KUKA KRL program: filwin69start.src

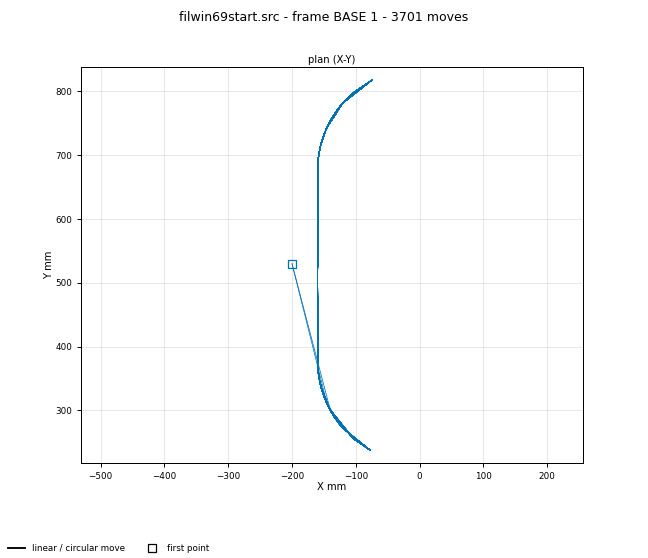
[picture p0: tool path of filwin69start.src in frame BASE 1, 3701 of 3702 moves have a stored position in this frame; points joined in program order, loops and branches not executed]
&ACCESS RVEO
&REL 11
&PARAM TEMPLATE = C:\KRC\Roboter\Template\vorgabe
&PARAM EDITMASK = *
DEF variable_helical2( )
;FOLD INI
  ;FOLD BASISTECH INI
    GLOBAL INTERRUPT DECL 3 WHEN $STOPMESS==TRUE DO IR_STOPM ( )
    INTERRUPT ON 3
    BAS (#INITMOV,0 )
  ;ENDFOLD (BASISTECH INI)
 ;FOLD USER INI


    ;Make your modifications here
  ;ENDFOLD (USER INI)
;ENDFOLD (INI)
ACTION(#AXIS_RESET,34,1000,#NOERROR,ERROR_CODE)
;FOLD PTP HOME  Vel= 100 % DEFAULT;%{PE}%MKUKATPBASIS,%CMOVE,%VPTP,%P 1:PTP, 2:HOME, 3:, 5:100, 7:DEFAULT
$BWDSTART = FALSE
PDAT_ACT=PDEFAULT
FDAT_ACT=FHOME
BAS (#PTP_PARAMS,100 )
$H_POS=XHOME
PTP  XHOME
;ENDFOLD
BAS(#TOOL,1)
BAS(#BASE,1)
$VEL_AXIS[1]=100
$VEL_AXIS[2]=100
$VEL_AXIS[3]=100
$VEL_AXIS[4]=100
$VEL_AXIS[5]=100
$VEL_AXIS[6]=100
$VEL_EXTAX[1]=100
$VEL_EXTAX[2]=100

$ACC_AXIS[1]=100
$ACC_AXIS[2]=100
$ACC_AXIS[3]=100
$ACC_AXIS[4]=100
$ACC_AXIS[5]=100
$ACC_AXIS[6]=100
$ACC_EXTAX[1]=100
$ACC_EXTAX[2]=100

;;;;;;;;; postprocessing parameters (date 2024-01-29T17:39:48.607859)
; qxconst: -159.99
; qxconstarcys: -152.5,146.5
; qE3offset: 0.00
; qyoffset: 530.00
; qswitchsplit: 3
; qthinningtol: 0.2010
;;;;;;;;;

SLIN {X  -200.000, Y  +530.000, Z    +0.000, A    +0.000, E1    +0.000, E3    +0.000, E4    +0.000}

SLIN {X  -139.652, Y  +299.435, Z    +0.000, E1   +73.041, E3  -288.222}
HALT
SPLINE
SPL {X  -136.475, Y  +294.006, Z    +0.000, E1   +72.670, E3  -282.347}
SPL {X  -133.214, Y  +288.895, Z    +0.000, E1   +72.272, E3  -276.699}
SPL {X  -129.829, Y  +284.006, Z    +0.000, E1   +71.844, E3  -271.224}
SPL {X  -126.314, Y  +279.309, Z    +0.000, E1   +71.374, E3  -265.932}
SPL {X  -122.705, Y  +274.834, Z    +0.000, E1   +70.869, E3  -260.920}
SPL {X  -119.804, Y  +271.463, Z    +0.000, E1   +70.429, E3  -257.202}
SPL {X   -77.409, Y  +237.483, Z    +0.000, E1   +59.013, E3  -163.526}
ENDSPLINE

SPLINE
SPL {X  -103.775, Y  +255.731, Z    +0.000, E1   +56.205, E3   +33.187}
SPL {X  -133.021, Y  +288.605, Z    +0.000, E1   +53.007, E3   +64.644}
SPL {X  -149.384, Y  +320.219, Z    +0.000, E1   +43.953, E3   +76.367}
SPL {X  -157.534, Y  +349.577, Z    +0.000, E1   +27.748, E3   +81.719}
SPL {X  -159.460, Y  +364.489, Z    +0.000, E1   +15.407, E3   +83.014}
SPL {X  -159.962, Y  +374.520, Z    +0.000, E1    +5.534, E3   +83.410}
SPL {X  -159.990, Y  +379.490, Z    +0.000, E1    +0.023, E3   +83.468}
SPL {X  -159.990, Y  +381.667, Z    +0.000, E1    -4.707, E3   +83.490}
SPL {X  -159.990, Y  +387.434, Z    +0.000, E1   -19.600, E3   +83.672}
SPL {X  -159.990, Y  +392.971, Z    +0.000, E1   -33.903, E3   +84.005}
SPL {X  -159.990, Y  +399.006, Z    +0.000, E1   -45.565, E3   +84.581}
SPL {X  -159.990, Y  +410.008, Z    +0.000, E1   -58.546, E3   +86.192}
SPL {X  -159.990, Y  +426.664, Z    +0.000, E1   -66.963, E3   +89.813}
SPL {X  -159.990, Y  +494.829, Z    +0.000, E1   -73.764, E3  +111.577}
SPL {X  -158.798, Y  +695.991, Z    +0.000, E1   -74.986, E3  +201.510}
SPL {X  -156.512, Y  +709.677, Z    +0.000, E1   -74.772, E3  +211.653}
SPL {X  -153.684, Y  +720.975, Z    +0.000, E1   -74.508, E3  +220.940}
SPL {X  -149.353, Y  +733.863, Z    +0.000, E1   -74.100, E3  +232.528}
SPL {X  -145.190, Y  +743.705, Z    +0.000, E1   -73.640, E3  +242.209}
SPL {X  -141.940, Y  +750.322, Z    +0.000, E1   -73.290, E3  +248.976}
SPL {X  -138.555, Y  +756.496, Z    +0.000, E1   -72.905, E3  +255.541}
SPL {X  -135.025, Y  +762.319, Z    +0.000, E1   -72.483, E3  +261.921}
SPL {X  -131.747, Y  +767.272, Z    +0.000, E1   -72.071, E3  +267.446}
SPL {X  -128.648, Y  +771.613, Z    +0.000, E1   -71.666, E3  +272.338}
SPL {X  -125.012, Y  +776.344, Z    +0.000, E1   -71.184, E3  +277.650}
SPL {X  -121.578, Y  +780.498, Z    +0.000, E1   -70.681, E3  +282.293}
SPL {X  -119.460, Y  +782.925, Z    +0.000, E1   -70.353, E3  +284.957}
SPL {X   -74.295, Y  +818.193, Z    +0.000, E1   -57.793, E3  +393.618}
ENDSPLINE

SPLINE
SPL {X  -120.240, Y  +782.043, Z    +0.000, E1   -55.019, E3  +592.114}
SPL {X  -145.777, Y  +742.423, Z    +0.000, E1   -46.722, E3  +613.993}
SPL {X  -154.920, Y  +716.458, Z    +0.000, E1   -35.175, E3  +620.048}
SPL {X  -159.063, Y  +693.702, Z    +0.000, E1   -19.028, E3  +622.830}
SPL {X  -159.958, Y  +679.684, Z    +0.000, E1    -5.688, E3  +623.541}
SPL {X  -159.990, Y  +674.512, Z    +0.000, E1    -0.026, E3  +623.606}
SPL {X  -159.990, Y  +672.767, Z    +0.000, E1    +3.705, E3  +623.619}
SPL {X  -159.990, Y  +669.310, Z    +0.000, E1   +12.444, E3  +623.693}
SPL {X  -159.990, Y  +665.511, Z    +0.000, E1   +22.359, E3  +623.852}
SPL {X  -159.990, Y  +658.432, Z    +0.000, E1   +38.720, E3  +624.377}
SPL {X  -159.990, Y  +646.280, Z    +0.000, E1   +56.156, E3  +625.906}
SPL {X  -159.990, Y  +625.549, Z    +0.000, E1   +67.208, E3  +630.427}
SPL {X  -159.990, Y  +550.186, Z    +0.000, E1   +73.637, E3  +655.833}
SPL {X  -159.493, Y  +364.902, Z    +0.000, E1   +74.541, E3  +742.826}
SPL {X  -156.915, Y  +346.281, Z    +0.000, E1   +74.304, E3  +756.422}
ENDSPLINE

SPLINE
SPL {X  -159.697, Y  +367.814, Z    +0.000, E1   +71.217, E3  +773.741}
ENDSPLINE

SPLINE
SPL {X  -157.536, Y  +349.586, Z    +0.000, E1   +71.787, E3  +781.039}
SPL {X  -154.855, Y  +337.291, Z    +0.000, E1   +72.155, E3  +785.793}
SPL {X  -150.925, Y  +324.412, Z    +0.000, E1   +72.419, E3  +791.687}
SPL {X  -146.819, Y  +313.931, Z    +0.000, E1   +72.621, E3  +796.380}
SPL {X  -140.820, Y  +301.561, Z    +0.000, E1   +73.023, E3  +800.297}
SPL {X  -136.475, Y  +294.006, Z    +0.000, E1   +72.670, E3  +807.206}
SPL {X  -133.214, Y  +288.895, Z    +0.000, E1   +72.272, E3  +812.853}
SPL {X  -129.829, Y  +284.006, Z    +0.000, E1   +71.844, E3  +818.328}
SPL {X  -126.314, Y  +279.309, Z    +0.000, E1   +71.374, E3  +823.621}
SPL {X  -122.705, Y  +274.834, Z    +0.000, E1   +70.869, E3  +828.632}
SPL {X  -119.804, Y  +271.463, Z    +0.000, E1   +70.429, E3  +832.351}
SPL {X   -77.409, Y  +237.483, Z    +0.000, E1   +59.013, E3  +926.026}
ENDSPLINE

SPLINE
SPL {X  -103.775, Y  +255.731, Z    +0.000, E1   +56.205, E3 +1122.739}
SPL {X  -141.196, Y  +302.265, Z    +0.000, E1   +49.914, E3 +1160.224}
SPL {X  -155.405, Y  +339.473, Z    +0.000, E1   +34.418, E3 +1169.925}
SPL {X  -159.172, Y  +361.346, Z    +0.000, E1   +18.323, E3 +1172.349}
SPL {X  -159.962, Y  +374.520, Z    +0.000, E1    +5.534, E3 +1172.962}
SPL {X  -159.990, Y  +379.490, Z    +0.000, E1    +0.023, E3 +1173.020}
SPL {X  -159.990, Y  +381.667, Z    +0.000, E1    -4.707, E3 +1173.042}
SPL {X  -159.990, Y  +385.814, Z    +0.000, E1   -15.621, E3 +1173.146}
SPL {X  -159.990, Y  +390.948, Z    +0.000, E1   -28.850, E3 +1173.422}
SPL {X  -159.990, Y  +399.006, Z    +0.000, E1   -45.565, E3 +1174.134}
SPL {X  -159.990, Y  +410.008, Z    +0.000, E1   -58.546, E3 +1175.744}
SPL {X  -159.990, Y  +426.664, Z    +0.000, E1   -66.963, E3 +1179.365}
SPL {X  -159.990, Y  +494.829, Z    +0.000, E1   -73.764, E3 +1201.129}
SPL {X  -158.798, Y  +695.991, Z    +0.000, E1   -74.986, E3 +1291.062}
SPL {X  -156.512, Y  +709.677, Z    +0.000, E1   -74.772, E3 +1301.205}
SPL {X  -153.684, Y  +720.975, Z    +0.000, E1   -74.508, E3 +1310.493}
SPL {X  -149.353, Y  +733.863, Z    +0.000, E1   -74.100, E3 +1322.080}
SPL {X  -145.190, Y  +743.705, Z    +0.000, E1   -73.640, E3 +1331.761}
SPL {X  -141.940, Y  +750.322, Z    +0.000, E1   -73.290, E3 +1338.528}
SPL {X  -138.555, Y  +756.496, Z    +0.000, E1   -72.905, E3 +1345.093}
SPL {X  -135.025, Y  +762.319, Z    +0.000, E1   -72.483, E3 +1351.473}
SPL {X  -131.747, Y  +767.272, Z    +0.000, E1   -72.071, E3 +1356.998}
SPL {X  -128.648, Y  +771.613, Z    +0.000, E1   -71.666, E3 +1361.890}
SPL {X  -125.012, Y  +776.344, Z    +0.000, E1   -71.184, E3 +1367.202}
SPL {X  -121.578, Y  +780.498, Z    +0.000, E1   -70.681, E3 +1371.845}
SPL {X  -119.460, Y  +782.925, Z    +0.000, E1   -70.353, E3 +1374.509}
SPL {X   -74.295, Y  +818.193, Z    +0.000, E1   -57.793, E3 +1483.170}
ENDSPLINE

SPLINE
SPL {X  -120.240, Y  +782.043, Z    +0.000, E1   -55.019, E3 +1681.666}
SPL {X  -145.777, Y  +742.423, Z    +0.000, E1   -46.722, E3 +1703.545}
SPL {X  -154.920, Y  +716.458, Z    +0.000, E1   -35.175, E3 +1709.600}
SPL {X  -159.063, Y  +693.702, Z    +0.000, E1   -19.028, E3 +1712.382}
SPL {X  -159.958, Y  +679.684, Z    +0.000, E1    -5.688, E3 +1713.094}
SPL {X  -159.990, Y  +674.512, Z    +0.000, E1    -0.026, E3 +1713.158}
SPL {X  -159.990, Y  +672.767, Z    +0.000, E1    +3.705, E3 +1713.172}
SPL {X  -159.990, Y  +669.310, Z    +0.000, E1   +12.444, E3 +1713.246}
SPL {X  -159.990, Y  +665.511, Z    +0.000, E1   +22.359, E3 +1713.404}
SPL {X  -159.990, Y  +658.432, Z    +0.000, E1   +38.720, E3 +1713.929}
SPL {X  -159.990, Y  +646.280, Z    +0.000, E1   +56.156, E3 +1715.458}
SPL {X  -159.990, Y  +625.549, Z    +0.000, E1   +67.208, E3 +1719.979}
SPL {X  -159.990, Y  +550.186, Z    +0.000, E1   +73.637, E3 +1745.385}
SPL {X  -159.493, Y  +364.902, Z    +0.000, E1   +74.541, E3 +1832.378}
SPL {X  -156.915, Y  +346.281, Z    +0.000, E1   +74.304, E3 +1845.974}
ENDSPLINE

SPLINE
SPL {X  -159.697, Y  +367.814, Z    +0.000, E1   +71.217, E3 +1863.293}
ENDSPLINE

SPLINE
SPL {X  -157.536, Y  +349.586, Z    +0.000, E1   +71.787, E3 +1870.591}
SPL {X  -154.855, Y  +337.291, Z    +0.000, E1   +72.155, E3 +1875.345}
SPL {X  -150.925, Y  +324.412, Z    +0.000, E1   +72.419, E3 +1881.239}
SPL {X  -146.819, Y  +313.931, Z    +0.000, E1   +72.621, E3 +1885.933}
SPL {X  -140.820, Y  +301.561, Z    +0.000, E1   +73.023, E3 +1889.849}
SPL {X  -136.475, Y  +294.006, Z    +0.000, E1   +72.670, E3 +1896.758}
SPL {X  -133.214, Y  +288.895, Z    +0.000, E1   +72.272, E3 +1902.406}
SPL {X  -129.829, Y  +284.006, Z    +0.000, E1   +71.844, E3 +1907.881}
SPL {X  -126.314, Y  +279.309, Z    +0.000, E1   +71.374, E3 +1913.173}
SPL {X  -122.705, Y  +274.834, Z    +0.000, E1   +70.869, E3 +1918.184}
SPL {X  -119.804, Y  +271.463, Z    +0.000, E1   +70.429, E3 +1921.903}
SPL {X   -77.409, Y  +237.483, Z    +0.000, E1   +59.013, E3 +2015.578}
ENDSPLINE

SPLINE
SPL {X  -103.775, Y  +255.731, Z    +0.000, E1   +56.205, E3 +2212.292}
SPL {X  -141.196, Y  +302.265, Z    +0.000, E1   +49.914, E3 +2249.777}
SPL {X  -155.405, Y  +339.473, Z    +0.000, E1   +34.418, E3 +2259.477}
SPL {X  -159.172, Y  +361.346, Z    +0.000, E1   +18.323, E3 +2261.902}
SPL {X  -159.962, Y  +374.520, Z    +0.000, E1    +5.534, E3 +2262.515}
SPL {X  -159.990, Y  +379.490, Z    +0.000, E1    +0.023, E3 +2262.572}
SPL {X  -159.990, Y  +381.667, Z    +0.000, E1    -4.707, E3 +2262.594}
SPL {X  -159.990, Y  +385.814, Z    +0.000, E1   -15.621, E3 +2262.698}
SPL {X  -159.990, Y  +390.948, Z    +0.000, E1   -28.850, E3 +2262.974}
SPL {X  -159.990, Y  +399.006, Z    +0.000, E1   -45.565, E3 +2263.686}
SPL {X  -159.990, Y  +410.008, Z    +0.000, E1   -58.546, E3 +2265.296}
SPL {X  -159.990, Y  +426.664, Z    +0.000, E1   -66.963, E3 +2268.917}
SPL {X  -159.990, Y  +494.829, Z    +0.000, E1   -73.764, E3 +2290.681}
SPL {X  -158.798, Y  +695.991, Z    +0.000, E1   -74.986, E3 +2380.614}
SPL {X  -156.512, Y  +709.677, Z    +0.000, E1   -74.772, E3 +2390.758}
SPL {X  -153.684, Y  +720.975, Z    +0.000, E1   -74.508, E3 +2400.045}
SPL {X  -150.879, Y  +729.719, Z    +0.000, E1   -74.224, E3 +2407.839}
SPL {X  -148.237, Y  +736.689, Z    +0.000, E1   -73.960, E3 +2414.393}
SPL {X  -145.190, Y  +743.705, Z    +0.000, E1   -73.640, E3 +2421.314}
SPL {X  -141.940, Y  +750.322, Z    +0.000, E1   -73.290, E3 +2428.081}
SPL {X  -138.555, Y  +756.496, Z    +0.000, E1   -72.905, E3 +2434.646}
SPL {X  -135.025, Y  +762.319, Z    +0.000, E1   -72.483, E3 +2441.025}
SPL {X  -131.747, Y  +767.272, Z    +0.000, E1   -72.071, E3 +2446.550}
SPL {X  -127.432, Y  +773.236, Z    +0.000, E1   -71.530, E3 +2453.236}
SPL {X  -124.036, Y  +777.554, Z    +0.000, E1   -71.026, E3 +2458.134}
SPL {X  -120.782, Y  +781.422, Z    +0.000, E1   -70.584, E3 +2462.392}
SPL {X   -74.295, Y  +818.193, Z    +0.000, E1   -57.793, E3 +2572.722}
ENDSPLINE

SPLINE
SPL {X  -105.102, Y  +797.125, Z    +0.000, E1   -55.734, E3 +2752.089}
SPL {X  -126.361, Y  +774.631, Z    +0.000, E1   -54.192, E3 +2777.757}
SPL {X  -145.777, Y  +742.423, Z    +0.000, E1   -46.722, E3 +2793.098}
SPL {X  -154.920, Y  +716.458, Z    +0.000, E1   -35.175, E3 +2799.153}
SPL {X  -159.063, Y  +693.702, Z    +0.000, E1   -19.028, E3 +2801.934}
SPL {X  -159.958, Y  +679.684, Z    +0.000, E1    -5.688, E3 +2802.646}
SPL {X  -159.990, Y  +674.512, Z    +0.000, E1    -0.026, E3 +2802.711}
SPL {X  -159.990, Y  +672.767, Z    +0.000, E1    +3.705, E3 +2802.724}
SPL {X  -159.990, Y  +669.310, Z    +0.000, E1   +12.444, E3 +2802.798}
SPL {X  -159.990, Y  +665.511, Z    +0.000, E1   +22.359, E3 +2802.957}
SPL {X  -159.990, Y  +660.776, Z    +0.000, E1   +34.018, E3 +2803.263}
SPL {X  -159.990, Y  +655.863, Z    +0.000, E1   +43.768, E3 +2803.721}
SPL {X  -159.990, Y  +646.280, Z    +0.000, E1   +56.156, E3 +2805.010}
SPL {X  -159.990, Y  +625.549, Z    +0.000, E1   +67.208, E3 +2809.532}
SPL {X  -159.990, Y  +550.186, Z    +0.000, E1   +73.637, E3 +2834.937}
SPL {X  -159.493, Y  +364.902, Z    +0.000, E1   +74.541, E3 +2921.931}
SPL {X  -156.915, Y  +346.281, Z    +0.000, E1   +74.304, E3 +2935.527}
ENDSPLINE

SPLINE
SPL {X  -159.697, Y  +367.814, Z    +0.000, E1   +71.217, E3 +2952.845}
ENDSPLINE

SPLINE
SPL {X  -157.536, Y  +349.586, Z    +0.000, E1   +71.787, E3 +2960.143}
SPL {X  -154.855, Y  +337.291, Z    +0.000, E1   +72.155, E3 +2964.897}
SPL {X  -150.925, Y  +324.412, Z    +0.000, E1   +72.419, E3 +2970.792}
SPL {X  -146.819, Y  +313.931, Z    +0.000, E1   +72.621, E3 +2975.485}
SPL {X  -140.820, Y  +301.561, Z    +0.000, E1   +73.023, E3 +2979.401}
SPL {X  -136.475, Y  +294.006, Z    +0.000, E1   +72.670, E3 +2986.310}
SPL {X  -133.214, Y  +288.895, Z    +0.000, E1   +72.272, E3 +2991.958}
SPL {X  -129.829, Y  +284.006, Z    +0.000, E1   +71.844, E3 +2997.433}
SPL {X  -126.314, Y  +279.309, Z    +0.000, E1   +71.374, E3 +3002.725}
SPL {X  -122.705, Y  +274.834, Z    +0.000, E1   +70.869, E3 +3007.736}
SPL {X  -119.804, Y  +271.463, Z    +0.000, E1   +70.429, E3 +3011.455}
SPL {X   -77.409, Y  +237.483, Z    +0.000, E1   +59.013, E3 +3105.131}
ENDSPLINE

SPLINE
SPL {X  -103.775, Y  +255.731, Z    +0.000, E1   +56.205, E3 +3301.844}
SPL {X  -141.196, Y  +302.265, Z    +0.000, E1   +49.914, E3 +3339.329}
SPL {X  -155.405, Y  +339.473, Z    +0.000, E1   +34.418, E3 +3349.029}
SPL {X  -159.172, Y  +361.346, Z    +0.000, E1   +18.323, E3 +3351.454}
SPL {X  -159.962, Y  +374.520, Z    +0.000, E1    +5.534, E3 +3352.067}
SPL {X  -159.990, Y  +379.490, Z    +0.000, E1    +0.023, E3 +3352.124}
SPL {X  -159.990, Y  +381.667, Z    +0.000, E1    -4.707, E3 +3352.146}
SPL {X  -159.990, Y  +387.434, Z    +0.000, E1   -19.600, E3 +3352.329}
SPL {X  -159.990, Y  +395.000, Z    +0.000, E1   -38.121, E3 +3352.838}
SPL {X  -159.990, Y  +406.380, Z    +0.000, E1   -55.108, E3 +3354.279}
SPL {X  -159.990, Y  +426.664, Z    +0.000, E1   -66.963, E3 +3358.469}
SPL {X  -159.990, Y  +494.829, Z    +0.000, E1   -73.764, E3 +3380.234}
SPL {X  -158.798, Y  +695.991, Z    +0.000, E1   -74.986, E3 +3470.166}
SPL {X  -156.512, Y  +709.677, Z    +0.000, E1   -74.772, E3 +3480.310}
SPL {X  -153.684, Y  +720.975, Z    +0.000, E1   -74.508, E3 +3489.597}
SPL {X  -149.353, Y  +733.863, Z    +0.000, E1   -74.100, E3 +3501.185}
SPL {X  -145.190, Y  +743.705, Z    +0.000, E1   -73.640, E3 +3510.866}
SPL {X  -141.940, Y  +750.322, Z    +0.000, E1   -73.290, E3 +3517.633}
SPL {X  -138.555, Y  +756.496, Z    +0.000, E1   -72.905, E3 +3524.198}
SPL {X  -135.025, Y  +762.319, Z    +0.000, E1   -72.483, E3 +3530.577}
SPL {X  -131.747, Y  +767.272, Z    +0.000, E1   -72.071, E3 +3536.102}
SPL {X  -127.432, Y  +773.236, Z    +0.000, E1   -71.530, E3 +3542.788}
SPL {X  -124.036, Y  +777.554, Z    +0.000, E1   -71.026, E3 +3547.686}
SPL {X  -120.782, Y  +781.422, Z    +0.000, E1   -70.584, E3 +3551.944}
SPL {X   -74.295, Y  +818.193, Z    +0.000, E1   -57.793, E3 +3662.275}
ENDSPLINE

SPLINE
SPL {X  -105.102, Y  +797.125, Z    +0.000, E1   -55.734, E3 +3841.641}
SPL {X  -126.361, Y  +774.631, Z    +0.000, E1   -54.192, E3 +3867.309}
SPL {X  -145.777, Y  +742.423, Z    +0.000, E1   -46.722, E3 +3882.650}
SPL {X  -154.920, Y  +716.458, Z    +0.000, E1   -35.175, E3 +3888.705}
SPL {X  -159.063, Y  +693.702, Z    +0.000, E1   -19.028, E3 +3891.486}
SPL {X  -159.958, Y  +679.684, Z    +0.000, E1    -5.688, E3 +3892.198}
SPL {X  -159.990, Y  +674.512, Z    +0.000, E1    -0.026, E3 +3892.263}
SPL {X  -159.990, Y  +672.767, Z    +0.000, E1    +3.705, E3 +3892.276}
SPL {X  -159.990, Y  +669.310, Z    +0.000, E1   +12.444, E3 +3892.350}
SPL {X  -159.990, Y  +665.511, Z    +0.000, E1   +22.359, E3 +3892.509}
SPL {X  -159.990, Y  +660.776, Z    +0.000, E1   +34.018, E3 +3892.815}
SPL {X  -159.990, Y  +655.863, Z    +0.000, E1   +43.768, E3 +3893.273}
SPL {X  -159.990, Y  +646.280, Z    +0.000, E1   +56.156, E3 +3894.562}
SPL {X  -159.990, Y  +625.549, Z    +0.000, E1   +67.208, E3 +3899.084}
SPL {X  -159.990, Y  +550.186, Z    +0.000, E1   +73.637, E3 +3924.490}
SPL {X  -159.493, Y  +364.902, Z    +0.000, E1   +74.541, E3 +4011.483}
SPL {X  -156.915, Y  +346.281, Z    +0.000, E1   +74.304, E3 +4025.079}
ENDSPLINE

SPLINE
SPL {X  -159.697, Y  +367.814, Z    +0.000, E1   +71.217, E3 +4042.397}
ENDSPLINE

SPLINE
SPL {X  -157.536, Y  +349.586, Z    +0.000, E1   +71.787, E3 +4049.696}
SPL {X  -154.855, Y  +337.291, Z    +0.000, E1   +72.155, E3 +4054.450}
SPL {X  -150.925, Y  +324.412, Z    +0.000, E1   +72.419, E3 +4060.344}
SPL {X  -146.819, Y  +313.931, Z    +0.000, E1   +72.621, E3 +4065.037}
SPL {X  -140.820, Y  +301.561, Z    +0.000, E1   +73.023, E3 +4068.953}
SPL {X  -136.475, Y  +294.006, Z    +0.000, E1   +72.670, E3 +4075.862}
SPL {X  -133.214, Y  +288.895, Z    +0.000, E1   +72.272, E3 +4081.510}
SPL {X  -129.829, Y  +284.006, Z    +0.000, E1   +71.844, E3 +4086.985}
SPL {X  -126.314, Y  +279.309, Z    +0.000, E1   +71.374, E3 +4092.277}
SPL {X  -122.705, Y  +274.834, Z    +0.000, E1   +70.869, E3 +4097.289}
SPL {X  -119.804, Y  +271.463, Z    +0.000, E1   +70.429, E3 +4101.007}
SPL {X   -77.409, Y  +237.483, Z    +0.000, E1   +59.013, E3 +4194.683}
ENDSPLINE

SPLINE
SPL {X  -103.775, Y  +255.731, Z    +0.000, E1   +56.205, E3 +4391.396}
SPL {X  -141.196, Y  +302.265, Z    +0.000, E1   +49.914, E3 +4428.881}
SPL {X  -155.405, Y  +339.473, Z    +0.000, E1   +34.418, E3 +4438.582}
SPL {X  -159.172, Y  +361.346, Z    +0.000, E1   +18.323, E3 +4441.006}
SPL {X  -159.962, Y  +374.520, Z    +0.000, E1    +5.534, E3 +4441.619}
SPL {X  -159.990, Y  +379.490, Z    +0.000, E1    +0.023, E3 +4441.677}
SPL {X  -159.990, Y  +381.667, Z    +0.000, E1    -4.707, E3 +4441.698}
SPL {X  -159.990, Y  +387.434, Z    +0.000, E1   -19.600, E3 +4441.881}
SPL {X  -159.990, Y  +395.000, Z    +0.000, E1   -38.121, E3 +4442.390}
SPL {X  -159.990, Y  +406.380, Z    +0.000, E1   -55.108, E3 +4443.832}
SPL {X  -159.990, Y  +426.664, Z    +0.000, E1   -66.963, E3 +4448.022}
SPL {X  -159.990, Y  +494.829, Z    +0.000, E1   -73.764, E3 +4469.786}
SPL {X  -158.798, Y  +695.991, Z    +0.000, E1   -74.986, E3 +4559.718}
SPL {X  -156.512, Y  +709.677, Z    +0.000, E1   -74.772, E3 +4569.862}
SPL {X  -153.684, Y  +720.975, Z    +0.000, E1   -74.508, E3 +4579.149}
SPL {X  -149.353, Y  +733.863, Z    +0.000, E1   -74.100, E3 +4590.737}
SPL {X  -145.190, Y  +743.705, Z    +0.000, E1   -73.640, E3 +4600.418}
SPL {X  -141.940, Y  +750.322, Z    +0.000, E1   -73.290, E3 +4607.185}
SPL {X  -138.555, Y  +756.496, Z    +0.000, E1   -72.905, E3 +4613.750}
SPL {X  -135.025, Y  +762.319, Z    +0.000, E1   -72.483, E3 +4620.130}
SPL {X  -131.747, Y  +767.272, Z    +0.000, E1   -72.071, E3 +4625.655}
SPL {X  -127.432, Y  +773.236, Z    +0.000, E1   -71.530, E3 +4632.340}
SPL {X  -124.036, Y  +777.554, Z    +0.000, E1   -71.026, E3 +4637.238}
SPL {X  -120.782, Y  +781.422, Z    +0.000, E1   -70.584, E3 +4641.496}
SPL {X   -74.295, Y  +818.193, Z    +0.000, E1   -57.793, E3 +4751.827}
ENDSPLINE

SPLINE
SPL {X  -105.102, Y  +797.125, Z    +0.000, E1   -55.734, E3 +4931.194}
SPL {X  -126.361, Y  +774.631, Z    +0.000, E1   -54.192, E3 +4956.861}
SPL {X  -145.777, Y  +742.423, Z    +0.000, E1   -46.722, E3 +4972.202}
SPL {X  -154.920, Y  +716.458, Z    +0.000, E1   -35.175, E3 +4978.257}
SPL {X  -158.252, Y  +700.019, Z    +0.000, E1   -24.087, E3 +4980.509}
SPL {X  -159.434, Y  +689.826, Z    +0.000, E1   -15.506, E3 +4981.327}
SPL {X  -159.958, Y  +679.684, Z    +0.000, E1    -5.688, E3 +4981.750}
SPL {X  -159.990, Y  +674.512, Z    +0.000, E1    -0.026, E3 +4981.815}
SPL {X  -159.990, Y  +672.767, Z    +0.000, E1    +3.705, E3 +4981.828}
SPL {X  -159.990, Y  +669.310, Z    +0.000, E1   +12.444, E3 +4981.902}
SPL {X  -159.990, Y  +665.511, Z    +0.000, E1   +22.359, E3 +4982.061}
SPL {X  -159.990, Y  +660.776, Z    +0.000, E1   +34.018, E3 +4982.368}
SPL {X  -159.990, Y  +655.863, Z    +0.000, E1   +43.768, E3 +4982.825}
SPL {X  -159.990, Y  +646.280, Z    +0.000, E1   +56.156, E3 +4984.114}
SPL {X  -159.990, Y  +625.549, Z    +0.000, E1   +67.208, E3 +4988.636}
SPL {X  -159.990, Y  +550.186, Z    +0.000, E1   +73.637, E3 +5014.042}
SPL {X  -159.878, Y  +371.520, Z    +0.000, E1   +74.559, E3 +5096.804}
SPL {X  -159.109, Y  +360.737, Z    +0.000, E1   +74.490, E3 +5103.928}
SPL {X  -156.915, Y  +346.281, Z    +0.000, E1   +74.304, E3 +5114.631}
ENDSPLINE

SPLINE
SPL {X  -159.697, Y  +367.814, Z    +0.000, E1   +71.217, E3 +5131.950}
ENDSPLINE

SPLINE
SPL {X  -156.028, Y  +342.114, Z    +0.000, E1   +72.020, E3 +5142.103}
SPL {X  -150.925, Y  +324.412, Z    +0.000, E1   +72.419, E3 +5149.896}
SPL {X  -146.819, Y  +313.931, Z    +0.000, E1   +72.621, E3 +5154.589}
SPL {X  -140.820, Y  +301.561, Z    +0.000, E1   +73.023, E3 +5158.506}
SPL {X  -136.475, Y  +294.006, Z    +0.000, E1   +72.670, E3 +5165.415}
SPL {X  -133.214, Y  +288.895, Z    +0.000, E1   +72.272, E3 +5171.062}
SPL {X  -129.829, Y  +284.006, Z    +0.000, E1   +71.844, E3 +5176.537}
SPL {X  -125.428, Y  +278.179, Z    +0.000, E1   +71.273, E3 +5183.075}
SPL {X  -120.729, Y  +272.518, Z    +0.000, E1   +70.593, E3 +5189.384}
SPL {X   -77.409, Y  +237.483, Z    +0.000, E1   +59.013, E3 +5284.235}
ENDSPLINE

SPLINE
SPL {X  -103.775, Y  +255.731, Z    +0.000, E1   +56.205, E3 +5480.948}
SPL {X  -141.196, Y  +302.265, Z    +0.000, E1   +49.914, E3 +5518.433}
SPL {X  -155.405, Y  +339.473, Z    +0.000, E1   +34.418, E3 +5528.134}
SPL {X  -159.172, Y  +361.346, Z    +0.000, E1   +18.323, E3 +5530.558}
SPL {X  -159.962, Y  +374.520, Z    +0.000, E1    +5.534, E3 +5531.171}
SPL {X  -159.990, Y  +379.490, Z    +0.000, E1    +0.023, E3 +5531.229}
SPL {X  -159.990, Y  +381.667, Z    +0.000, E1    -4.707, E3 +5531.251}
SPL {X  -159.990, Y  +385.814, Z    +0.000, E1   -15.621, E3 +5531.355}
SPL {X  -159.990, Y  +390.948, Z    +0.000, E1   -28.850, E3 +5531.631}
SPL {X  -159.990, Y  +399.006, Z    +0.000, E1   -45.565, E3 +5532.342}
SPL {X  -159.990, Y  +410.008, Z    +0.000, E1   -58.546, E3 +5533.953}
SPL {X  -159.990, Y  +430.714, Z    +0.000, E1   -67.965, E3 +5538.758}
SPL {X  -159.990, Y  +500.758, Z    +0.000, E1   -73.927, E3 +5561.434}
SPL {X  -158.798, Y  +695.991, Z    +0.000, E1   -74.986, E3 +5649.271}
SPL {X  -156.512, Y  +709.677, Z    +0.000, E1   -74.772, E3 +5659.414}
SPL {X  -153.684, Y  +720.975, Z    +0.000, E1   -74.508, E3 +5668.702}
SPL {X  -149.353, Y  +733.863, Z    +0.000, E1   -74.100, E3 +5680.289}
SPL {X  -145.190, Y  +743.705, Z    +0.000, E1   -73.640, E3 +5689.970}
SPL {X  -141.940, Y  +750.322, Z    +0.000, E1   -73.290, E3 +5696.737}
SPL {X  -138.555, Y  +756.496, Z    +0.000, E1   -72.905, E3 +5703.302}
SPL {X  -135.025, Y  +762.319, Z    +0.000, E1   -72.483, E3 +5709.682}
SPL {X  -131.747, Y  +767.272, Z    +0.000, E1   -72.071, E3 +5715.207}
SPL {X  -128.648, Y  +771.613, Z    +0.000, E1   -71.666, E3 +5720.099}
SPL {X  -125.012, Y  +776.344, Z    +0.000, E1   -71.184, E3 +5725.411}
SPL {X  -120.782, Y  +781.422, Z    +0.000, E1   -70.584, E3 +5731.049}
SPL {X   -74.295, Y  +818.193, Z    +0.000, E1   -57.793, E3 +5841.379}
ENDSPLINE

SPLINE
SPL {X  -120.240, Y  +782.043, Z    +0.000, E1   -55.019, E3 +6039.875}
SPL {X  -145.777, Y  +742.423, Z    +0.000, E1   -46.722, E3 +6061.754}
SPL {X  -154.920, Y  +716.458, Z    +0.000, E1   -35.175, E3 +6067.809}
SPL {X  -158.252, Y  +700.019, Z    +0.000, E1   -24.087, E3 +6070.061}
SPL {X  -159.676, Y  +686.525, Z    +0.000, E1   -12.514, E3 +6071.051}
SPL {X  -159.990, Y  +674.678, Z    +0.000, E1    -0.382, E3 +6071.366}
SPL {X  -159.990, Y  +672.767, Z    +0.000, E1    +3.705, E3 +6071.381}
SPL {X  -159.990, Y  +669.310, Z    +0.000, E1   +12.444, E3 +6071.455}
SPL {X  -159.990, Y  +665.511, Z    +0.000, E1   +22.359, E3 +6071.613}
SPL {X  -159.990, Y  +658.432, Z    +0.000, E1   +38.720, E3 +6072.138}
SPL {X  -159.990, Y  +646.280, Z    +0.000, E1   +56.156, E3 +6073.667}
SPL {X  -159.990, Y  +625.549, Z    +0.000, E1   +67.208, E3 +6078.188}
SPL {X  -159.990, Y  +550.186, Z    +0.000, E1   +73.637, E3 +6103.594}
SPL {X  -159.493, Y  +364.902, Z    +0.000, E1   +74.541, E3 +6190.587}
SPL {X  -156.915, Y  +346.281, Z    +0.000, E1   +74.304, E3 +6204.183}
ENDSPLINE

SPLINE
SPL {X  -159.697, Y  +367.814, Z    +0.000, E1   +71.217, E3 +6221.502}
ENDSPLINE

SPLINE
SPL {X  -157.536, Y  +349.586, Z    +0.000, E1   +71.787, E3 +6228.800}
SPL {X  -154.855, Y  +337.291, Z    +0.000, E1   +72.155, E3 +6233.554}
SPL {X  -150.925, Y  +324.412, Z    +0.000, E1   +72.419, E3 +6239.448}
SPL {X  -146.819, Y  +313.931, Z    +0.000, E1   +72.621, E3 +6244.142}
SPL {X  -140.820, Y  +301.561, Z    +0.000, E1   +73.023, E3 +6248.058}
SPL {X  -136.475, Y  +294.006, Z    +0.000, E1   +72.670, E3 +6254.967}
SPL {X  -133.214, Y  +288.895, Z    +0.000, E1   +72.272, E3 +6260.615}
SPL {X  -129.829, Y  +284.006, Z    +0.000, E1   +71.844, E3 +6266.089}
SPL {X  -126.314, Y  +279.309, Z    +0.000, E1   +71.374, E3 +6271.382}
SPL {X  -122.705, Y  +274.834, Z    +0.000, E1   +70.869, E3 +6276.393}
SPL {X  -119.804, Y  +271.463, Z    +0.000, E1   +70.429, E3 +6280.112}
SPL {X   -77.409, Y  +237.483, Z    +0.000, E1   +59.013, E3 +6373.787}
ENDSPLINE

SPLINE
SPL {X  -103.775, Y  +255.731, Z    +0.000, E1   +56.205, E3 +6570.501}
SPL {X  -133.021, Y  +288.605, Z    +0.000, E1   +53.007, E3 +6601.957}
SPL {X  -149.384, Y  +320.219, Z    +0.000, E1   +43.953, E3 +6613.680}
SPL {X  -157.534, Y  +349.577, Z    +0.000, E1   +27.748, E3 +6619.032}
SPL {X  -159.460, Y  +364.489, Z    +0.000, E1   +15.407, E3 +6620.328}
SPL {X  -159.962, Y  +374.520, Z    +0.000, E1    +5.534, E3 +6620.724}
SPL {X  -159.990, Y  +379.490, Z    +0.000, E1    +0.023, E3 +6620.781}
SPL {X  -159.990, Y  +381.667, Z    +0.000, E1    -4.707, E3 +6620.803}
SPL {X  -159.990, Y  +387.434, Z    +0.000, E1   -19.600, E3 +6620.985}
SPL {X  -159.990, Y  +392.971, Z    +0.000, E1   -33.903, E3 +6621.318}
SPL {X  -159.990, Y  +399.006, Z    +0.000, E1   -45.565, E3 +6621.895}
SPL {X  -159.990, Y  +410.008, Z    +0.000, E1   -58.546, E3 +6623.505}
SPL {X  -159.990, Y  +426.664, Z    +0.000, E1   -66.963, E3 +6627.126}
SPL {X  -159.990, Y  +494.829, Z    +0.000, E1   -73.764, E3 +6648.890}
SPL {X  -158.798, Y  +695.991, Z    +0.000, E1   -74.986, E3 +6738.823}
SPL {X  -156.512, Y  +709.677, Z    +0.000, E1   -74.772, E3 +6748.967}
SPL {X  -153.684, Y  +720.975, Z    +0.000, E1   -74.508, E3 +6758.254}
SPL {X  -149.353, Y  +733.863, Z    +0.000, E1   -74.100, E3 +6769.842}
SPL {X  -145.190, Y  +743.705, Z    +0.000, E1   -73.640, E3 +6779.523}
SPL {X  -141.940, Y  +750.322, Z    +0.000, E1   -73.290, E3 +6786.290}
SPL {X  -138.555, Y  +756.496, Z    +0.000, E1   -72.905, E3 +6792.855}
SPL {X  -135.025, Y  +762.319, Z    +0.000, E1   -72.483, E3 +6799.234}
SPL {X  -131.747, Y  +767.272, Z    +0.000, E1   -72.071, E3 +6804.759}
SPL {X  -128.648, Y  +771.613, Z    +0.000, E1   -71.666, E3 +6809.651}
SPL {X  -125.012, Y  +776.344, Z    +0.000, E1   -71.184, E3 +6814.963}
SPL {X  -121.578, Y  +780.498, Z    +0.000, E1   -70.681, E3 +6819.606}
SPL {X  -119.460, Y  +782.925, Z    +0.000, E1   -70.353, E3 +6822.270}
SPL {X   -74.295, Y  +818.193, Z    +0.000, E1   -57.793, E3 +6930.931}
ENDSPLINE

SPLINE
SPL {X  -120.240, Y  +782.043, Z    +0.000, E1   -55.019, E3 +7129.427}
SPL {X  -145.777, Y  +742.423, Z    +0.000, E1   -46.722, E3 +7151.307}
SPL {X  -154.920, Y  +716.458, Z    +0.000, E1   -35.175, E3 +7157.362}
SPL {X  -159.063, Y  +693.702, Z    +0.000, E1   -19.028, E3 +7160.143}
SPL {X  -159.958, Y  +679.684, Z    +0.000, E1    -5.688, E3 +7160.855}
SPL {X  -159.990, Y  +674.512, Z    +0.000, E1    -0.026, E3 +7160.920}
SPL {X  -159.990, Y  +672.767, Z    +0.000, E1    +3.705, E3 +7160.933}
SPL {X  -159.990, Y  +669.310, Z    +0.000, E1   +12.444, E3 +7161.007}
SPL {X  -159.990, Y  +665.511, Z    +0.000, E1   +22.359, E3 +7161.166}
SPL {X  -159.990, Y  +658.432, Z    +0.000, E1   +38.720, E3 +7161.690}
SPL {X  -159.990, Y  +646.280, Z    +0.000, E1   +56.156, E3 +7163.219}
SPL {X  -159.990, Y  +625.549, Z    +0.000, E1   +67.208, E3 +7167.741}
SPL {X  -159.990, Y  +550.186, Z    +0.000, E1   +73.637, E3 +7193.146}
SPL {X  -159.878, Y  +371.520, Z    +0.000, E1   +74.559, E3 +7275.908}
SPL {X  -158.372, Y  +354.804, Z    +0.000, E1   +74.445, E3 +7287.213}
SPL {X  -156.009, Y  +342.031, Z    +0.000, E1   +74.195, E3 +7297.223}
ENDSPLINE

SPLINE
SPL {X  -159.697, Y  +367.814, Z    +0.000, E1   +71.217, E3 +7311.054}
ENDSPLINE

SPLINE
SPL {X  -156.028, Y  +342.114, Z    +0.000, E1   +72.020, E3 +7321.208}
SPL {X  -150.925, Y  +324.412, Z    +0.000, E1   +72.419, E3 +7329.001}
SPL {X  -144.972, Y  +309.824, Z    +0.000, E1   +72.799, E3 +7334.602}
SPL {X  -139.605, Y  +299.351, Z    +0.000, E1   +73.035, E3 +7338.734}
SPL {X  -136.475, Y  +294.006, Z    +0.000, E1   +72.670, E3 +7344.519}
SPL {X  -133.214, Y  +288.895, Z    +0.000, E1   +72.272, E3 +7350.167}
SPL {X  -129.829, Y  +284.006, Z    +0.000, E1   +71.844, E3 +7355.642}
SPL {X  -125.428, Y  +278.179, Z    +0.000, E1   +71.273, E3 +7362.179}
SPL {X  -120.729, Y  +272.518, Z    +0.000, E1   +70.593, E3 +7368.489}
SPL {X   -77.409, Y  +237.483, Z    +0.000, E1   +59.013, E3 +7463.340}
ENDSPLINE

SPLINE
SPL {X  -103.775, Y  +255.731, Z    +0.000, E1   +56.205, E3 +7660.053}
SPL {X  -133.021, Y  +288.605, Z    +0.000, E1   +53.007, E3 +7691.509}
SPL {X  -149.384, Y  +320.219, Z    +0.000, E1   +43.953, E3 +7703.233}
SPL {X  -157.534, Y  +349.577, Z    +0.000, E1   +27.748, E3 +7708.585}
SPL {X  -159.460, Y  +364.489, Z    +0.000, E1   +15.407, E3 +7709.880}
SPL {X  -159.962, Y  +374.520, Z    +0.000, E1    +5.534, E3 +7710.276}
SPL {X  -159.990, Y  +379.741, Z    +0.000, E1    -0.257, E3 +7710.335}
SPL {X  -159.990, Y  +384.604, Z    +0.000, E1   -12.124, E3 +7710.423}
SPL {X  -159.990, Y  +389.475, Z    +0.000, E1   -25.351, E3 +7710.637}
SPL {X  -159.990, Y  +395.000, Z    +0.000, E1   -38.121, E3 +7711.047}
SPL {X  -159.990, Y  +406.380, Z    +0.000, E1   -55.108, E3 +7712.488}
SPL {X  -159.990, Y  +426.664, Z    +0.000, E1   -66.963, E3 +7716.678}
SPL {X  -159.990, Y  +494.829, Z    +0.000, E1   -73.764, E3 +7738.443}
SPL {X  -158.798, Y  +695.991, Z    +0.000, E1   -74.986, E3 +7828.375}
SPL {X  -156.512, Y  +709.677, Z    +0.000, E1   -74.772, E3 +7838.519}
SPL {X  -153.684, Y  +720.975, Z    +0.000, E1   -74.508, E3 +7847.806}
SPL {X  -149.353, Y  +733.863, Z    +0.000, E1   -74.100, E3 +7859.394}
SPL {X  -145.190, Y  +743.705, Z    +0.000, E1   -73.640, E3 +7869.075}
SPL {X  -141.940, Y  +750.322, Z    +0.000, E1   -73.290, E3 +7875.842}
SPL {X  -138.555, Y  +756.496, Z    +0.000, E1   -72.905, E3 +7882.407}
SPL {X  -135.025, Y  +762.319, Z    +0.000, E1   -72.483, E3 +7888.786}
SPL {X  -131.747, Y  +767.272, Z    +0.000, E1   -72.071, E3 +7894.311}
SPL {X  -127.432, Y  +773.236, Z    +0.000, E1   -71.530, E3 +7900.997}
SPL {X  -124.036, Y  +777.554, Z    +0.000, E1   -71.026, E3 +7905.895}
SPL {X  -120.782, Y  +781.422, Z    +0.000, E1   -70.584, E3 +7910.153}
SPL {X   -74.295, Y  +818.193, Z    +0.000, E1   -57.793, E3 +8020.484}
ENDSPLINE

SPLINE
SPL {X  -120.240, Y  +782.043, Z    +0.000, E1   -55.019, E3 +8218.980}
SPL {X  -145.777, Y  +742.423, Z    +0.000, E1   -46.722, E3 +8240.859}
SPL {X  -154.920, Y  +716.458, Z    +0.000, E1   -35.175, E3 +8246.914}
SPL {X  -158.252, Y  +700.019, Z    +0.000, E1   -24.087, E3 +8249.166}
SPL {X  -159.676, Y  +686.525, Z    +0.000, E1   -12.514, E3 +8250.156}
SPL {X  -159.990, Y  +674.678, Z    +0.000, E1    -0.382, E3 +8250.471}
SPL {X  -159.990, Y  +672.767, Z    +0.000, E1    +3.705, E3 +8250.485}
SPL {X  -159.990, Y  +669.310, Z    +0.000, E1   +12.444, E3 +8250.559}
SPL {X  -159.990, Y  +665.511, Z    +0.000, E1   +22.359, E3 +8250.718}
SPL {X  -159.990, Y  +660.776, Z    +0.000, E1   +34.018, E3 +8251.024}
SPL {X  -159.990, Y  +655.863, Z    +0.000, E1   +43.768, E3 +8251.482}
SPL {X  -159.990, Y  +646.280, Z    +0.000, E1   +56.156, E3 +8252.771}
SPL {X  -159.990, Y  +625.549, Z    +0.000, E1   +67.208, E3 +8257.293}
SPL {X  -159.990, Y  +550.186, Z    +0.000, E1   +73.637, E3 +8282.699}
SPL {X  -159.878, Y  +371.520, Z    +0.000, E1   +74.559, E3 +8365.461}
SPL {X  -159.109, Y  +360.737, Z    +0.000, E1   +74.490, E3 +8372.585}
SPL {X  -156.915, Y  +346.281, Z    +0.000, E1   +74.304, E3 +8383.288}
ENDSPLINE

SPLINE
SPL {X  -159.697, Y  +367.814, Z    +0.000, E1   +71.217, E3 +8400.606}
ENDSPLINE

SPLINE
SPL {X  -156.028, Y  +342.114, Z    +0.000, E1   +72.020, E3 +8410.760}
SPL {X  -150.925, Y  +324.412, Z    +0.000, E1   +72.419, E3 +8418.553}
SPL {X  -146.819, Y  +313.931, Z    +0.000, E1   +72.621, E3 +8423.246}
SPL {X  -140.820, Y  +301.561, Z    +0.000, E1   +73.023, E3 +8427.162}
SPL {X  -136.475, Y  +294.006, Z    +0.000, E1   +72.670, E3 +8434.071}
SPL {X  -133.214, Y  +288.895, Z    +0.000, E1   +72.272, E3 +8439.719}
SPL {X  -129.829, Y  +284.006, Z    +0.000, E1   +71.844, E3 +8445.194}
SPL {X  -125.428, Y  +278.179, Z    +0.000, E1   +71.273, E3 +8451.731}
SPL {X  -120.729, Y  +272.518, Z    +0.000, E1   +70.593, E3 +8458.041}
SPL {X   -77.409, Y  +237.483, Z    +0.000, E1   +59.013, E3 +8552.892}
ENDSPLINE

SPLINE
SPL {X  -103.775, Y  +255.731, Z    +0.000, E1   +56.205, E3 +8749.605}
SPL {X  -141.196, Y  +302.265, Z    +0.000, E1   +49.914, E3 +8787.090}
SPL {X  -155.405, Y  +339.473, Z    +0.000, E1   +34.418, E3 +8796.791}
SPL {X  -159.172, Y  +361.346, Z    +0.000, E1   +18.323, E3 +8799.215}
SPL {X  -159.962, Y  +374.520, Z    +0.000, E1    +5.534, E3 +8799.828}
SPL {X  -159.990, Y  +379.490, Z    +0.000, E1    +0.023, E3 +8799.886}
SPL {X  -159.990, Y  +381.667, Z    +0.000, E1    -4.707, E3 +8799.907}
SPL {X  -159.990, Y  +385.814, Z    +0.000, E1   -15.621, E3 +8800.011}
SPL {X  -159.990, Y  +390.948, Z    +0.000, E1   -28.850, E3 +8800.288}
SPL {X  -159.990, Y  +399.006, Z    +0.000, E1   -45.565, E3 +8800.999}
SPL {X  -159.990, Y  +410.008, Z    +0.000, E1   -58.546, E3 +8802.610}
SPL {X  -159.990, Y  +426.664, Z    +0.000, E1   -66.963, E3 +8806.231}
SPL {X  -159.990, Y  +494.829, Z    +0.000, E1   -73.764, E3 +8827.995}
SPL {X  -158.798, Y  +695.991, Z    +0.000, E1   -74.986, E3 +8917.927}
SPL {X  -156.512, Y  +709.677, Z    +0.000, E1   -74.772, E3 +8928.071}
SPL {X  -153.684, Y  +720.975, Z    +0.000, E1   -74.508, E3 +8937.358}
SPL {X  -149.353, Y  +733.863, Z    +0.000, E1   -74.100, E3 +8948.946}
SPL {X  -145.190, Y  +743.705, Z    +0.000, E1   -73.640, E3 +8958.627}
SPL {X  -141.940, Y  +750.322, Z    +0.000, E1   -73.290, E3 +8965.394}
SPL {X  -138.555, Y  +756.496, Z    +0.000, E1   -72.905, E3 +8971.959}
SPL {X  -135.025, Y  +762.319, Z    +0.000, E1   -72.483, E3 +8978.339}
SPL {X  -131.747, Y  +767.272, Z    +0.000, E1   -72.071, E3 +8983.864}
SPL {X  -128.648, Y  +771.613, Z    +0.000, E1   -71.666, E3 +8988.756}
SPL {X  -125.012, Y  +776.344, Z    +0.000, E1   -71.184, E3 +8994.067}
SPL {X  -121.578, Y  +780.498, Z    +0.000, E1   -70.681, E3 +8998.711}
SPL {X  -119.460, Y  +782.925, Z    +0.000, E1   -70.353, E3 +9001.375}
SPL {X   -74.295, Y  +818.193, Z    +0.000, E1   -57.793, E3 +9110.036}
ENDSPLINE

SPLINE
SPL {X  -120.240, Y  +782.043, Z    +0.000, E1   -55.019, E3 +9308.532}
SPL {X  -145.777, Y  +742.423, Z    +0.000, E1   -46.722, E3 +9330.411}
SPL {X  -154.920, Y  +716.458, Z    +0.000, E1   -35.175, E3 +9336.466}
SPL {X  -159.063, Y  +693.702, Z    +0.000, E1   -19.028, E3 +9339.248}
SPL {X  -159.958, Y  +679.684, Z    +0.000, E1    -5.688, E3 +9339.959}
SPL {X  -159.990, Y  +674.512, Z    +0.000, E1    -0.026, E3 +9340.024}
SPL {X  -159.990, Y  +672.767, Z    +0.000, E1    +3.705, E3 +9340.037}
SPL {X  -159.990, Y  +669.310, Z    +0.000, E1   +12.444, E3 +9340.111}
SPL {X  -159.990, Y  +665.511, Z    +0.000, E1   +22.359, E3 +9340.270}
SPL {X  -159.990, Y  +658.432, Z    +0.000, E1   +38.720, E3 +9340.795}
SPL {X  -159.990, Y  +646.280, Z    +0.000, E1   +56.156, E3 +9342.323}
SPL {X  -159.990, Y  +625.549, Z    +0.000, E1   +67.208, E3 +9346.845}
SPL {X  -159.990, Y  +550.186, Z    +0.000, E1   +73.637, E3 +9372.251}
SPL {X  -159.493, Y  +364.902, Z    +0.000, E1   +74.541, E3 +9459.244}
SPL {X  -156.915, Y  +346.281, Z    +0.000, E1   +74.304, E3 +9472.840}
ENDSPLINE

SPLINE
SPL {X  -159.697, Y  +367.814, Z    +0.000, E1   +71.217, E3 +9490.159}
ENDSPLINE

SPLINE
SPL {X  -156.028, Y  +342.114, Z    +0.000, E1   +72.020, E3 +9500.312}
SPL {X  -150.925, Y  +324.412, Z    +0.000, E1   +72.419, E3 +9508.105}
SPL {X  -144.972, Y  +309.824, Z    +0.000, E1   +72.799, E3 +9513.707}
SPL {X  -139.605, Y  +299.351, Z    +0.000, E1   +73.035, E3 +9517.839}
SPL {X  -136.475, Y  +294.006, Z    +0.000, E1   +72.670, E3 +9523.624}
SPL {X  -133.214, Y  +288.895, Z    +0.000, E1   +72.272, E3 +9529.271}
SPL {X  -129.829, Y  +284.006, Z    +0.000, E1   +71.844, E3 +9534.746}
SPL {X  -126.314, Y  +279.309, Z    +0.000, E1   +71.374, E3 +9540.039}
SPL {X  -122.705, Y  +274.834, Z    +0.000, E1   +70.869, E3 +9545.050}
SPL {X  -119.804, Y  +271.463, Z    +0.000, E1   +70.429, E3 +9548.768}
SPL {X   -77.409, Y  +237.483, Z    +0.000, E1   +59.013, E3 +9642.444}
ENDSPLINE

SPLINE
SPL {X  -103.775, Y  +255.731, Z    +0.000, E1   +56.205, E3 +9839.157}
SPL {X  -133.021, Y  +288.605, Z    +0.000, E1   +53.007, E3 +9870.614}
SPL {X  -149.384, Y  +320.219, Z    +0.000, E1   +43.953, E3 +9882.337}
SPL {X  -157.534, Y  +349.577, Z    +0.000, E1   +27.748, E3 +9887.689}
SPL {X  -159.460, Y  +364.489, Z    +0.000, E1   +15.407, E3 +9888.985}
SPL {X  -159.962, Y  +374.520, Z    +0.000, E1    +5.534, E3 +9889.380}
SPL {X  -159.990, Y  +379.490, Z    +0.000, E1    +0.023, E3 +9889.438}
SPL {X  -159.990, Y  +381.667, Z    +0.000, E1    -4.707, E3 +9889.460}
SPL {X  -159.990, Y  +387.434, Z    +0.000, E1   -19.600, E3 +9889.642}
SPL {X  -159.990, Y  +392.971, Z    +0.000, E1   -33.903, E3 +9889.975}
SPL {X  -159.990, Y  +399.006, Z    +0.000, E1   -45.565, E3 +9890.551}
SPL {X  -159.990, Y  +410.008, Z    +0.000, E1   -58.546, E3 +9892.162}
SPL {X  -159.990, Y  +426.664, Z    +0.000, E1   -66.963, E3 +9895.783}
SPL {X  -159.990, Y  +494.829, Z    +0.000, E1   -73.764, E3 +9917.547}
SPL {X  -158.798, Y  +695.991, Z    +0.000, E1   -74.986, E3 +10007.480}
SPL {X  -156.512, Y  +709.677, Z    +0.000, E1   -74.772, E3 +10017.623}
SPL {X  -153.684, Y  +720.975, Z    +0.000, E1   -74.508, E3 +10026.911}
SPL {X  -149.353, Y  +733.863, Z    +0.000, E1   -74.100, E3 +10038.498}
SPL {X  -145.190, Y  +743.705, Z    +0.000, E1   -73.640, E3 +10048.179}
SPL {X  -141.940, Y  +750.322, Z    +0.000, E1   -73.290, E3 +10054.946}
SPL {X  -138.555, Y  +756.496, Z    +0.000, E1   -72.905, E3 +10061.511}
SPL {X  -135.025, Y  +762.319, Z    +0.000, E1   -72.483, E3 +10067.891}
SPL {X  -131.747, Y  +767.272, Z    +0.000, E1   -72.071, E3 +10073.416}
SPL {X  -127.432, Y  +773.236, Z    +0.000, E1   -71.530, E3 +10080.101}
SPL {X  -124.036, Y  +777.554, Z    +0.000, E1   -71.026, E3 +10085.000}
SPL {X  -120.782, Y  +781.422, Z    +0.000, E1   -70.584, E3 +10089.258}
SPL {X   -74.295, Y  +818.193, Z    +0.000, E1   -57.793, E3 +10199.588}
ENDSPLINE

SPLINE
SPL {X  -105.102, Y  +797.125, Z    +0.000, E1   -55.734, E3 +10378.955}
SPL {X  -126.361, Y  +774.631, Z    +0.000, E1   -54.192, E3 +10404.622}
SPL {X  -145.777, Y  +742.423, Z    +0.000, E1   -46.722, E3 +10419.963}
SPL {X  -154.920, Y  +716.458, Z    +0.000, E1   -35.175, E3 +10426.018}
SPL {X  -159.063, Y  +693.702, Z    +0.000, E1   -19.028, E3 +10428.800}
SPL {X  -159.958, Y  +679.684, Z    +0.000, E1    -5.688, E3 +10429.512}
SPL {X  -159.990, Y  +674.512, Z    +0.000, E1    -0.026, E3 +10429.576}
SPL {X  -159.990, Y  +672.767, Z    +0.000, E1    +3.705, E3 +10429.590}
SPL {X  -159.990, Y  +669.310, Z    +0.000, E1   +12.444, E3 +10429.664}
SPL {X  -159.990, Y  +665.511, Z    +0.000, E1   +22.359, E3 +10429.822}
SPL {X  -159.990, Y  +660.776, Z    +0.000, E1   +34.018, E3 +10430.129}
SPL {X  -159.990, Y  +655.863, Z    +0.000, E1   +43.768, E3 +10430.586}
SPL {X  -159.990, Y  +646.280, Z    +0.000, E1   +56.156, E3 +10431.876}
SPL {X  -159.990, Y  +625.549, Z    +0.000, E1   +67.208, E3 +10436.397}
SPL {X  -159.990, Y  +550.186, Z    +0.000, E1   +73.637, E3 +10461.803}
SPL {X  -159.493, Y  +364.902, Z    +0.000, E1   +74.541, E3 +10548.796}
SPL {X  -156.915, Y  +346.281, Z    +0.000, E1   +74.304, E3 +10562.392}
ENDSPLINE

SPLINE
SPL {X  -159.697, Y  +367.814, Z    +0.000, E1   +71.217, E3 +10579.711}
ENDSPLINE

SPLINE
SPL {X  -157.536, Y  +349.586, Z    +0.000, E1   +71.787, E3 +10587.009}
SPL {X  -154.855, Y  +337.291, Z    +0.000, E1   +72.155, E3 +10591.763}
SPL {X  -150.925, Y  +324.412, Z    +0.000, E1   +72.419, E3 +10597.657}
SPL {X  -146.819, Y  +313.931, Z    +0.000, E1   +72.621, E3 +10602.351}
SPL {X  -140.820, Y  +301.561, Z    +0.000, E1   +73.023, E3 +10606.267}
SPL {X  -136.475, Y  +294.006, Z    +0.000, E1   +72.670, E3 +10613.176}
SPL {X  -133.214, Y  +288.895, Z    +0.000, E1   +72.272, E3 +10618.824}
SPL {X  -129.829, Y  +284.006, Z    +0.000, E1   +71.844, E3 +10624.298}
SPL {X  -126.314, Y  +279.309, Z    +0.000, E1   +71.374, E3 +10629.591}
SPL {X  -122.705, Y  +274.834, Z    +0.000, E1   +70.869, E3 +10634.602}
SPL {X  -119.804, Y  +271.463, Z    +0.000, E1   +70.429, E3 +10638.321}
SPL {X   -77.409, Y  +237.483, Z    +0.000, E1   +59.013, E3 +10731.996}
ENDSPLINE

SPLINE
SPL {X  -103.775, Y  +255.731, Z    +0.000, E1   +56.205, E3 +10928.710}
SPL {X  -141.196, Y  +302.265, Z    +0.000, E1   +49.914, E3 +10966.195}
SPL {X  -155.405, Y  +339.473, Z    +0.000, E1   +34.418, E3 +10975.895}
SPL {X  -159.172, Y  +361.346, Z    +0.000, E1   +18.323, E3 +10978.320}
SPL {X  -159.962, Y  +374.520, Z    +0.000, E1    +5.534, E3 +10978.933}
SPL {X  -159.990, Y  +379.490, Z    +0.000, E1    +0.023, E3 +10978.990}
SPL {X  -159.990, Y  +381.667, Z    +0.000, E1    -4.707, E3 +10979.012}
SPL {X  -159.990, Y  +387.434, Z    +0.000, E1   -19.600, E3 +10979.194}
SPL {X  -159.990, Y  +395.000, Z    +0.000, E1   -38.121, E3 +10979.703}
SPL {X  -159.990, Y  +406.380, Z    +0.000, E1   -55.108, E3 +10981.145}
SPL {X  -159.990, Y  +426.664, Z    +0.000, E1   -66.963, E3 +10985.335}
SPL {X  -159.990, Y  +494.829, Z    +0.000, E1   -73.764, E3 +11007.099}
SPL {X  -158.798, Y  +695.991, Z    +0.000, E1   -74.986, E3 +11097.032}
SPL {X  -156.512, Y  +709.677, Z    +0.000, E1   -74.772, E3 +11107.175}
SPL {X  -153.684, Y  +720.975, Z    +0.000, E1   -74.508, E3 +11116.463}
SPL {X  -149.353, Y  +733.863, Z    +0.000, E1   -74.100, E3 +11128.051}
SPL {X  -145.190, Y  +743.705, Z    +0.000, E1   -73.640, E3 +11137.732}
SPL {X  -141.940, Y  +750.322, Z    +0.000, E1   -73.290, E3 +11144.498}
SPL {X  -138.555, Y  +756.496, Z    +0.000, E1   -72.905, E3 +11151.063}
SPL {X  -135.025, Y  +762.319, Z    +0.000, E1   -72.483, E3 +11157.443}
SPL {X  -131.747, Y  +767.272, Z    +0.000, E1   -72.071, E3 +11162.968}
SPL {X  -127.432, Y  +773.236, Z    +0.000, E1   -71.530, E3 +11169.653}
SPL {X  -124.036, Y  +777.554, Z    +0.000, E1   -71.026, E3 +11174.552}
SPL {X  -120.782, Y  +781.422, Z    +0.000, E1   -70.584, E3 +11178.810}
SPL {X   -74.295, Y  +818.193, Z    +0.000, E1   -57.793, E3 +11289.140}
ENDSPLINE

SPLINE
SPL {X  -105.102, Y  +797.125, Z    +0.000, E1   -55.734, E3 +11468.507}
SPL {X  -126.361, Y  +774.631, Z    +0.000, E1   -54.192, E3 +11494.175}
SPL {X  -145.777, Y  +742.423, Z    +0.000, E1   -46.722, E3 +11509.516}
SPL {X  -154.920, Y  +716.458, Z    +0.000, E1   -35.175, E3 +11515.571}
SPL {X  -158.252, Y  +700.019, Z    +0.000, E1   -24.087, E3 +11517.822}
SPL {X  -159.434, Y  +689.826, Z    +0.000, E1   -15.506, E3 +11518.641}
SPL {X  -159.958, Y  +679.684, Z    +0.000, E1    -5.688, E3 +11519.064}
SPL {X  -159.990, Y  +674.512, Z    +0.000, E1    -0.026, E3 +11519.129}
SPL {X  -159.990, Y  +672.767, Z    +0.000, E1    +3.705, E3 +11519.142}
SPL {X  -159.990, Y  +669.310, Z    +0.000, E1   +12.444, E3 +11519.216}
SPL {X  -159.990, Y  +665.511, Z    +0.000, E1   +22.359, E3 +11519.375}
SPL {X  -159.990, Y  +660.776, Z    +0.000, E1   +34.018, E3 +11519.681}
SPL {X  -159.990, Y  +655.863, Z    +0.000, E1   +43.768, E3 +11520.139}
SPL {X  -159.990, Y  +646.280, Z    +0.000, E1   +56.156, E3 +11521.428}
SPL {X  -159.990, Y  +625.549, Z    +0.000, E1   +67.208, E3 +11525.950}
SPL {X  -159.990, Y  +550.186, Z    +0.000, E1   +73.637, E3 +11551.355}
SPL {X  -159.878, Y  +371.520, Z    +0.000, E1   +74.559, E3 +11634.117}
SPL {X  -159.109, Y  +360.737, Z    +0.000, E1   +74.490, E3 +11641.242}
SPL {X  -156.915, Y  +346.281, Z    +0.000, E1   +74.304, E3 +11651.945}
ENDSPLINE

SPLINE
SPL {X  -159.697, Y  +367.814, Z    +0.000, E1   +71.217, E3 +11669.263}
ENDSPLINE

SPLINE
SPL {X  -156.028, Y  +342.114, Z    +0.000, E1   +72.020, E3 +11679.417}
SPL {X  -150.925, Y  +324.412, Z    +0.000, E1   +72.419, E3 +11687.209}
SPL {X  -146.819, Y  +313.931, Z    +0.000, E1   +72.621, E3 +11691.903}
SPL {X  -140.820, Y  +301.561, Z    +0.000, E1   +73.023, E3 +11695.819}
SPL {X  -136.475, Y  +294.006, Z    +0.000, E1   +72.670, E3 +11702.728}
SPL {X  -133.214, Y  +288.895, Z    +0.000, E1   +72.272, E3 +11708.376}
SPL {X  -129.829, Y  +284.006, Z    +0.000, E1   +71.844, E3 +11713.851}
SPL {X  -125.428, Y  +278.179, Z    +0.000, E1   +71.273, E3 +11720.388}
SPL {X  -120.729, Y  +272.518, Z    +0.000, E1   +70.593, E3 +11726.698}
SPL {X   -77.409, Y  +237.483, Z    +0.000, E1   +59.013, E3 +11821.549}
ENDSPLINE

SPLINE
SPL {X  -103.775, Y  +255.731, Z    +0.000, E1   +56.205, E3 +12018.262}
SPL {X  -141.196, Y  +302.265, Z    +0.000, E1   +49.914, E3 +12055.747}
SPL {X  -155.405, Y  +339.473, Z    +0.000, E1   +34.418, E3 +12065.447}
SPL {X  -159.172, Y  +361.346, Z    +0.000, E1   +18.323, E3 +12067.872}
SPL {X  -159.962, Y  +374.520, Z    +0.000, E1    +5.534, E3 +12068.485}
SPL {X  -159.990, Y  +379.490, Z    +0.000, E1    +0.023, E3 +12068.542}
SPL {X  -159.990, Y  +381.667, Z    +0.000, E1    -4.707, E3 +12068.564}
SPL {X  -159.990, Y  +385.814, Z    +0.000, E1   -15.621, E3 +12068.668}
SPL {X  -159.990, Y  +390.948, Z    +0.000, E1   -28.850, E3 +12068.944}
SPL {X  -159.990, Y  +399.006, Z    +0.000, E1   -45.565, E3 +12069.656}
SPL {X  -159.990, Y  +410.008, Z    +0.000, E1   -58.546, E3 +12071.266}
SPL {X  -159.990, Y  +430.714, Z    +0.000, E1   -67.965, E3 +12076.071}
SPL {X  -159.990, Y  +500.758, Z    +0.000, E1   -73.927, E3 +12098.747}
SPL {X  -158.798, Y  +695.991, Z    +0.000, E1   -74.986, E3 +12186.584}
SPL {X  -156.512, Y  +709.677, Z    +0.000, E1   -74.772, E3 +12196.728}
SPL {X  -153.684, Y  +720.975, Z    +0.000, E1   -74.508, E3 +12206.015}
SPL {X  -150.879, Y  +729.719, Z    +0.000, E1   -74.224, E3 +12213.809}
SPL {X  -148.237, Y  +736.689, Z    +0.000, E1   -73.960, E3 +12220.363}
SPL {X  -145.190, Y  +743.705, Z    +0.000, E1   -73.640, E3 +12227.284}
SPL {X  -141.940, Y  +750.322, Z    +0.000, E1   -73.290, E3 +12234.051}
SPL {X  -138.555, Y  +756.496, Z    +0.000, E1   -72.905, E3 +12240.616}
SPL {X  -135.025, Y  +762.319, Z    +0.000, E1   -72.483, E3 +12246.995}
SPL {X  -131.747, Y  +767.272, Z    +0.000, E1   -72.071, E3 +12252.520}
SPL {X  -127.432, Y  +773.236, Z    +0.000, E1   -71.530, E3 +12259.206}
SPL {X  -124.036, Y  +777.554, Z    +0.000, E1   -71.026, E3 +12264.104}
SPL {X  -120.782, Y  +781.422, Z    +0.000, E1   -70.584, E3 +12268.362}
SPL {X   -74.295, Y  +818.193, Z    +0.000, E1   -57.793, E3 +12378.693}
ENDSPLINE

SPLINE
SPL {X  -105.102, Y  +797.125, Z    +0.000, E1   -55.734, E3 +12558.059}
SPL {X  -126.361, Y  +774.631, Z    +0.000, E1   -54.192, E3 +12583.727}
SPL {X  -145.777, Y  +742.423, Z    +0.000, E1   -46.722, E3 +12599.068}
SPL {X  -154.920, Y  +716.458, Z    +0.000, E1   -35.175, E3 +12605.123}
SPL {X  -158.252, Y  +700.019, Z    +0.000, E1   -24.087, E3 +12607.375}
SPL {X  -159.676, Y  +686.525, Z    +0.000, E1   -12.514, E3 +12608.365}
SPL {X  -159.990, Y  +674.678, Z    +0.000, E1    -0.382, E3 +12608.680}
SPL {X  -159.990, Y  +672.767, Z    +0.000, E1    +3.705, E3 +12608.694}
SPL {X  -159.990, Y  +669.310, Z    +0.000, E1   +12.444, E3 +12608.768}
SPL {X  -159.990, Y  +665.511, Z    +0.000, E1   +22.359, E3 +12608.927}
SPL {X  -159.990, Y  +658.432, Z    +0.000, E1   +38.720, E3 +12609.452}
SPL {X  -159.990, Y  +646.280, Z    +0.000, E1   +56.156, E3 +12610.980}
SPL {X  -159.990, Y  +625.549, Z    +0.000, E1   +67.208, E3 +12615.502}
SPL {X  -159.990, Y  +550.186, Z    +0.000, E1   +73.637, E3 +12640.908}
SPL {X  -159.493, Y  +364.902, Z    +0.000, E1   +74.541, E3 +12727.901}
SPL {X  -156.915, Y  +346.281, Z    +0.000, E1   +74.304, E3 +12741.497}
ENDSPLINE

SPLINE
SPL {X  -159.697, Y  +367.814, Z    +0.000, E1   +71.217, E3 +12758.815}
ENDSPLINE

SPLINE
SPL {X  -156.028, Y  +342.114, Z    +0.000, E1   +72.020, E3 +12768.969}
SPL {X  -150.925, Y  +324.412, Z    +0.000, E1   +72.419, E3 +12776.762}
SPL {X  -144.972, Y  +309.824, Z    +0.000, E1   +72.799, E3 +12782.364}
SPL {X  -139.605, Y  +299.351, Z    +0.000, E1   +73.035, E3 +12786.495}
SPL {X  -136.475, Y  +294.006, Z    +0.000, E1   +72.670, E3 +12792.280}
SPL {X  -133.214, Y  +288.895, Z    +0.000, E1   +72.272, E3 +12797.928}
SPL {X  -129.829, Y  +284.006, Z    +0.000, E1   +71.844, E3 +12803.403}
SPL {X  -126.314, Y  +279.309, Z    +0.000, E1   +71.374, E3 +12808.695}
SPL {X  -122.705, Y  +274.834, Z    +0.000, E1   +70.869, E3 +12813.706}
SPL {X  -119.804, Y  +271.463, Z    +0.000, E1   +70.429, E3 +12817.425}
SPL {X   -77.409, Y  +237.483, Z    +0.000, E1   +59.013, E3 +12911.101}
ENDSPLINE

SPLINE
SPL {X  -103.775, Y  +255.731, Z    +0.000, E1   +56.205, E3 +13107.814}
SPL {X  -133.021, Y  +288.605, Z    +0.000, E1   +53.007, E3 +13139.270}
SPL {X  -149.384, Y  +320.219, Z    +0.000, E1   +43.953, E3 +13150.994}
SPL {X  -157.534, Y  +349.577, Z    +0.000, E1   +27.748, E3 +13156.346}
SPL {X  -159.460, Y  +364.489, Z    +0.000, E1   +15.407, E3 +13157.641}
SPL {X  -159.962, Y  +374.520, Z    +0.000, E1    +5.534, E3 +13158.037}
SPL {X  -159.990, Y  +379.490, Z    +0.000, E1    +0.023, E3 +13158.094}
SPL {X  -159.990, Y  +381.667, Z    +0.000, E1    -4.707, E3 +13158.116}
SPL {X  -159.990, Y  +387.434, Z    +0.000, E1   -19.600, E3 +13158.299}
SPL {X  -159.990, Y  +392.971, Z    +0.000, E1   -33.903, E3 +13158.632}
SPL {X  -159.990, Y  +399.006, Z    +0.000, E1   -45.565, E3 +13159.208}
SPL {X  -159.990, Y  +410.008, Z    +0.000, E1   -58.546, E3 +13160.818}
SPL {X  -159.990, Y  +426.664, Z    +0.000, E1   -66.963, E3 +13164.440}
SPL {X  -159.990, Y  +494.829, Z    +0.000, E1   -73.764, E3 +13186.204}
SPL {X  -158.798, Y  +695.991, Z    +0.000, E1   -74.986, E3 +13276.136}
SPL {X  -156.512, Y  +709.677, Z    +0.000, E1   -74.772, E3 +13286.280}
SPL {X  -153.684, Y  +720.975, Z    +0.000, E1   -74.508, E3 +13295.567}
SPL {X  -149.353, Y  +733.863, Z    +0.000, E1   -74.100, E3 +13307.155}
SPL {X  -145.190, Y  +743.705, Z    +0.000, E1   -73.640, E3 +13316.836}
SPL {X  -141.940, Y  +750.322, Z    +0.000, E1   -73.290, E3 +13323.603}
SPL {X  -138.555, Y  +756.496, Z    +0.000, E1   -72.905, E3 +13330.168}
SPL {X  -135.025, Y  +762.319, Z    +0.000, E1   -72.483, E3 +13336.548}
SPL {X  -131.747, Y  +767.272, Z    +0.000, E1   -72.071, E3 +13342.073}
SPL {X  -128.648, Y  +771.613, Z    +0.000, E1   -71.666, E3 +13346.965}
SPL {X  -125.012, Y  +776.344, Z    +0.000, E1   -71.184, E3 +13352.276}
SPL {X  -121.578, Y  +780.498, Z    +0.000, E1   -70.681, E3 +13356.920}
SPL {X  -119.460, Y  +782.925, Z    +0.000, E1   -70.353, E3 +13359.584}
SPL {X   -74.295, Y  +818.193, Z    +0.000, E1   -57.793, E3 +13468.245}
ENDSPLINE

SPLINE
SPL {X  -120.240, Y  +782.043, Z    +0.000, E1   -55.019, E3 +13666.741}
SPL {X  -145.777, Y  +742.423, Z    +0.000, E1   -46.722, E3 +13688.620}
SPL {X  -154.920, Y  +716.458, Z    +0.000, E1   -35.175, E3 +13694.675}
SPL {X  -159.063, Y  +693.702, Z    +0.000, E1   -19.028, E3 +13697.456}
SPL {X  -159.958, Y  +679.684, Z    +0.000, E1    -5.688, E3 +13698.168}
SPL {X  -159.990, Y  +674.512, Z    +0.000, E1    -0.026, E3 +13698.233}
SPL {X  -159.990, Y  +672.767, Z    +0.000, E1    +3.705, E3 +13698.246}
SPL {X  -159.990, Y  +669.310, Z    +0.000, E1   +12.444, E3 +13698.320}
SPL {X  -159.990, Y  +665.511, Z    +0.000, E1   +22.359, E3 +13698.479}
SPL {X  -159.990, Y  +658.432, Z    +0.000, E1   +38.720, E3 +13699.004}
SPL {X  -159.990, Y  +646.280, Z    +0.000, E1   +56.156, E3 +13700.532}
SPL {X  -159.990, Y  +625.549, Z    +0.000, E1   +67.208, E3 +13705.054}
SPL {X  -159.990, Y  +550.186, Z    +0.000, E1   +73.637, E3 +13730.460}
SPL {X  -159.878, Y  +371.520, Z    +0.000, E1   +74.559, E3 +13813.222}
SPL {X  -159.109, Y  +360.737, Z    +0.000, E1   +74.490, E3 +13820.346}
SPL {X  -156.915, Y  +346.281, Z    +0.000, E1   +74.304, E3 +13831.049}
ENDSPLINE

SPLINE
SPL {X  -159.697, Y  +367.814, Z    +0.000, E1   +71.217, E3 +13848.368}
ENDSPLINE

SPLINE
SPL {X  -157.536, Y  +349.586, Z    +0.000, E1   +71.787, E3 +13855.666}
SPL {X  -154.855, Y  +337.291, Z    +0.000, E1   +72.155, E3 +13860.420}
SPL {X  -150.925, Y  +324.412, Z    +0.000, E1   +72.419, E3 +13866.314}
SPL {X  -146.819, Y  +313.931, Z    +0.000, E1   +72.621, E3 +13871.007}
SPL {X  -140.820, Y  +301.561, Z    +0.000, E1   +73.023, E3 +13874.924}
SPL {X  -136.475, Y  +294.006, Z    +0.000, E1   +72.670, E3 +13881.833}
SPL {X  -133.214, Y  +288.895, Z    +0.000, E1   +72.272, E3 +13887.480}
SPL {X  -129.829, Y  +284.006, Z    +0.000, E1   +71.844, E3 +13892.955}
SPL {X  -126.314, Y  +279.309, Z    +0.000, E1   +71.374, E3 +13898.248}
SPL {X  -122.705, Y  +274.834, Z    +0.000, E1   +70.869, E3 +13903.259}
SPL {X  -119.804, Y  +271.463, Z    +0.000, E1   +70.429, E3 +13906.977}
SPL {X   -77.409, Y  +237.483, Z    +0.000, E1   +59.013, E3 +14000.653}
ENDSPLINE

SPLINE
SPL {X  -103.775, Y  +255.731, Z    +0.000, E1   +56.205, E3 +14197.366}
SPL {X  -141.196, Y  +302.265, Z    +0.000, E1   +49.914, E3 +14234.851}
SPL {X  -153.296, Y  +331.706, Z    +0.000, E1   +38.681, E3 +14243.270}
SPL {X  -157.534, Y  +349.577, Z    +0.000, E1   +27.748, E3 +14245.898}
SPL {X  -159.460, Y  +364.489, Z    +0.000, E1   +15.407, E3 +14247.194}
SPL {X  -159.962, Y  +374.520, Z    +0.000, E1    +5.534, E3 +14247.589}
SPL {X  -159.990, Y  +379.490, Z    +0.000, E1    +0.023, E3 +14247.647}
SPL {X  -159.990, Y  +381.667, Z    +0.000, E1    -4.707, E3 +14247.669}
SPL {X  -159.990, Y  +385.814, Z    +0.000, E1   -15.621, E3 +14247.772}
SPL {X  -159.990, Y  +390.948, Z    +0.000, E1   -28.850, E3 +14248.049}
SPL {X  -159.990, Y  +399.006, Z    +0.000, E1   -45.565, E3 +14248.760}
SPL {X  -159.990, Y  +410.008, Z    +0.000, E1   -58.546, E3 +14250.371}
SPL {X  -159.990, Y  +430.714, Z    +0.000, E1   -67.965, E3 +14255.176}
SPL {X  -159.990, Y  +500.758, Z    +0.000, E1   -73.927, E3 +14277.851}
SPL {X  -158.798, Y  +695.991, Z    +0.000, E1   -74.986, E3 +14365.689}
SPL {X  -156.512, Y  +709.677, Z    +0.000, E1   -74.772, E3 +14375.832}
SPL {X  -153.684, Y  +720.975, Z    +0.000, E1   -74.508, E3 +14385.120}
SPL {X  -150.879, Y  +729.719, Z    +0.000, E1   -74.224, E3 +14392.913}
SPL {X  -148.237, Y  +736.689, Z    +0.000, E1   -73.960, E3 +14399.467}
SPL {X  -145.190, Y  +743.705, Z    +0.000, E1   -73.640, E3 +14406.388}
SPL {X  -141.940, Y  +750.322, Z    +0.000, E1   -73.290, E3 +14413.155}
SPL {X  -138.555, Y  +756.496, Z    +0.000, E1   -72.905, E3 +14419.720}
SPL {X  -135.025, Y  +762.319, Z    +0.000, E1   -72.483, E3 +14426.100}
SPL {X  -131.747, Y  +767.272, Z    +0.000, E1   -72.071, E3 +14431.625}
SPL {X  -127.432, Y  +773.236, Z    +0.000, E1   -71.530, E3 +14438.310}
SPL {X  -124.036, Y  +777.554, Z    +0.000, E1   -71.026, E3 +14443.209}
SPL {X  -120.782, Y  +781.422, Z    +0.000, E1   -70.584, E3 +14447.467}
SPL {X   -74.295, Y  +818.193, Z    +0.000, E1   -57.793, E3 +14557.797}
ENDSPLINE

SPLINE
SPL {X  -120.240, Y  +782.043, Z    +0.000, E1   -55.019, E3 +14756.293}
SPL {X  -145.777, Y  +742.423, Z    +0.000, E1   -46.722, E3 +14778.172}
SPL {X  -154.920, Y  +716.458, Z    +0.000, E1   -35.175, E3 +14784.227}
SPL {X  -158.252, Y  +700.019, Z    +0.000, E1   -24.087, E3 +14786.479}
SPL {X  -159.676, Y  +686.525, Z    +0.000, E1   -12.514, E3 +14787.469}
SPL {X  -159.990, Y  +674.678, Z    +0.000, E1    -0.382, E3 +14787.784}
SPL {X  -159.990, Y  +672.767, Z    +0.000, E1    +3.705, E3 +14787.799}
SPL {X  -159.990, Y  +669.310, Z    +0.000, E1   +12.444, E3 +14787.873}
SPL {X  -159.990, Y  +665.511, Z    +0.000, E1   +22.359, E3 +14788.031}
SPL {X  -159.990, Y  +660.776, Z    +0.000, E1   +34.018, E3 +14788.338}
SPL {X  -159.990, Y  +655.863, Z    +0.000, E1   +43.768, E3 +14788.795}
SPL {X  -159.990, Y  +646.280, Z    +0.000, E1   +56.156, E3 +14790.085}
SPL {X  -159.990, Y  +625.549, Z    +0.000, E1   +67.208, E3 +14794.606}
SPL {X  -159.990, Y  +550.186, Z    +0.000, E1   +73.637, E3 +14820.012}
SPL {X  -159.878, Y  +371.520, Z    +0.000, E1   +74.559, E3 +14902.774}
SPL {X  -159.109, Y  +360.737, Z    +0.000, E1   +74.490, E3 +14909.898}
SPL {X  -156.915, Y  +346.281, Z    +0.000, E1   +74.304, E3 +14920.601}
ENDSPLINE

SPLINE
SPL {X  -159.697, Y  +367.814, Z    +0.000, E1   +71.217, E3 +14937.920}
ENDSPLINE

SPLINE
SPL {X  -157.536, Y  +349.586, Z    +0.000, E1   +71.787, E3 +14945.218}
SPL {X  -154.855, Y  +337.291, Z    +0.000, E1   +72.155, E3 +14949.972}
SPL {X  -150.925, Y  +324.412, Z    +0.000, E1   +72.419, E3 +14955.866}
SPL {X  -144.972, Y  +309.824, Z    +0.000, E1   +72.799, E3 +14961.468}
SPL {X  -139.605, Y  +299.351, Z    +0.000, E1   +73.035, E3 +14965.600}
SPL {X  -136.475, Y  +294.006, Z    +0.000, E1   +72.670, E3 +14971.385}
SPL {X  -133.214, Y  +288.895, Z    +0.000, E1   +72.272, E3 +14977.033}
SPL {X  -129.829, Y  +284.006, Z    +0.000, E1   +71.844, E3 +14982.507}
SPL {X  -126.314, Y  +279.309, Z    +0.000, E1   +71.374, E3 +14987.800}
SPL {X  -122.705, Y  +274.834, Z    +0.000, E1   +70.869, E3 +14992.811}
SPL {X  -119.804, Y  +271.463, Z    +0.000, E1   +70.429, E3 +14996.530}
SPL {X   -77.409, Y  +237.483, Z    +0.000, E1   +59.013, E3 +15090.205}
ENDSPLINE

SPLINE
SPL {X  -103.775, Y  +255.731, Z    +0.000, E1   +56.205, E3 +15286.919}
SPL {X  -141.196, Y  +302.265, Z    +0.000, E1   +49.914, E3 +15324.404}
SPL {X  -155.405, Y  +339.473, Z    +0.000, E1   +34.418, E3 +15334.104}
SPL {X  -158.399, Y  +354.990, Z    +0.000, E1   +23.559, E3 +15336.035}
SPL {X  -159.460, Y  +364.489, Z    +0.000, E1   +15.407, E3 +15336.746}
SPL {X  -159.962, Y  +374.520, Z    +0.000, E1    +5.534, E3 +15337.142}
SPL {X  -159.990, Y  +379.490, Z    +0.000, E1    +0.023, E3 +15337.199}
SPL {X  -159.990, Y  +381.667, Z    +0.000, E1    -4.707, E3 +15337.221}
SPL {X  -159.990, Y  +385.814, Z    +0.000, E1   -15.621, E3 +15337.325}
SPL {X  -159.990, Y  +390.948, Z    +0.000, E1   -28.850, E3 +15337.601}
SPL {X  -159.990, Y  +399.006, Z    +0.000, E1   -45.565, E3 +15338.313}
SPL {X  -159.990, Y  +410.008, Z    +0.000, E1   -58.546, E3 +15339.923}
SPL {X  -159.990, Y  +426.664, Z    +0.000, E1   -66.963, E3 +15343.544}
SPL {X  -159.990, Y  +494.829, Z    +0.000, E1   -73.764, E3 +15365.308}
SPL {X  -158.798, Y  +695.991, Z    +0.000, E1   -74.986, E3 +15455.241}
SPL {X  -156.512, Y  +709.677, Z    +0.000, E1   -74.772, E3 +15465.384}
SPL {X  -153.684, Y  +720.975, Z    +0.000, E1   -74.508, E3 +15474.672}
SPL {X  -149.353, Y  +733.863, Z    +0.000, E1   -74.100, E3 +15486.260}
SPL {X  -145.190, Y  +743.705, Z    +0.000, E1   -73.640, E3 +15495.941}
SPL {X  -141.940, Y  +750.322, Z    +0.000, E1   -73.290, E3 +15502.707}
SPL {X  -138.555, Y  +756.496, Z    +0.000, E1   -72.905, E3 +15509.272}
SPL {X  -135.025, Y  +762.319, Z    +0.000, E1   -72.483, E3 +15515.652}
SPL {X  -131.747, Y  +767.272, Z    +0.000, E1   -72.071, E3 +15521.177}
SPL {X  -128.648, Y  +771.613, Z    +0.000, E1   -71.666, E3 +15526.069}
SPL {X  -125.012, Y  +776.344, Z    +0.000, E1   -71.184, E3 +15531.381}
SPL {X  -120.782, Y  +781.422, Z    +0.000, E1   -70.584, E3 +15537.019}
SPL {X   -74.295, Y  +818.193, Z    +0.000, E1   -57.793, E3 +15647.349}
ENDSPLINE

SPLINE
SPL {X  -120.240, Y  +782.043, Z    +0.000, E1   -55.019, E3 +15845.845}
SPL {X  -145.777, Y  +742.423, Z    +0.000, E1   -46.722, E3 +15867.725}
SPL {X  -154.920, Y  +716.458, Z    +0.000, E1   -35.175, E3 +15873.780}
SPL {X  -159.063, Y  +693.702, Z    +0.000, E1   -19.028, E3 +15876.561}
SPL {X  -159.958, Y  +679.684, Z    +0.000, E1    -5.688, E3 +15877.273}
SPL {X  -159.990, Y  +674.512, Z    +0.000, E1    -0.026, E3 +15877.337}
SPL {X  -159.990, Y  +672.767, Z    +0.000, E1    +3.705, E3 +15877.351}
SPL {X  -159.990, Y  +669.310, Z    +0.000, E1   +12.444, E3 +15877.425}
SPL {X  -159.990, Y  +665.511, Z    +0.000, E1   +22.359, E3 +15877.583}
SPL {X  -159.990, Y  +658.432, Z    +0.000, E1   +38.720, E3 +15878.108}
SPL {X  -159.990, Y  +646.280, Z    +0.000, E1   +56.156, E3 +15879.637}
SPL {X  -159.990, Y  +625.549, Z    +0.000, E1   +67.208, E3 +15884.159}
SPL {X  -159.990, Y  +550.186, Z    +0.000, E1   +73.637, E3 +15909.564}
SPL {X  -159.493, Y  +364.902, Z    +0.000, E1   +74.541, E3 +15996.558}
SPL {X  -156.915, Y  +346.281, Z    +0.000, E1   +74.304, E3 +16010.154}
ENDSPLINE

SPLINE
SPL {X  -159.697, Y  +367.814, Z    +0.000, E1   +71.217, E3 +16027.472}
ENDSPLINE

SPLINE
SPL {X  -157.536, Y  +349.586, Z    +0.000, E1   +71.787, E3 +16034.770}
SPL {X  -154.855, Y  +337.291, Z    +0.000, E1   +72.155, E3 +16039.524}
SPL {X  -150.925, Y  +324.412, Z    +0.000, E1   +72.419, E3 +16045.418}
SPL {X  -144.972, Y  +309.824, Z    +0.000, E1   +72.799, E3 +16051.020}
SPL {X  -139.605, Y  +299.351, Z    +0.000, E1   +73.035, E3 +16055.152}
SPL {X  -136.475, Y  +294.006, Z    +0.000, E1   +72.670, E3 +16060.937}
SPL {X  -133.214, Y  +288.895, Z    +0.000, E1   +72.272, E3 +16066.585}
SPL {X  -129.829, Y  +284.006, Z    +0.000, E1   +71.844, E3 +16072.060}
SPL {X  -125.428, Y  +278.179, Z    +0.000, E1   +71.273, E3 +16078.597}
SPL {X  -120.729, Y  +272.518, Z    +0.000, E1   +70.593, E3 +16084.907}
SPL {X   -77.409, Y  +237.483, Z    +0.000, E1   +59.013, E3 +16179.757}
ENDSPLINE

SPLINE
SPL {X  -103.775, Y  +255.731, Z    +0.000, E1   +56.205, E3 +16376.471}
SPL {X  -141.196, Y  +302.265, Z    +0.000, E1   +49.914, E3 +16413.956}
SPL {X  -155.405, Y  +339.473, Z    +0.000, E1   +34.418, E3 +16423.656}
SPL {X  -159.172, Y  +361.346, Z    +0.000, E1   +18.323, E3 +16426.081}
SPL {X  -159.962, Y  +374.520, Z    +0.000, E1    +5.534, E3 +16426.694}
SPL {X  -159.990, Y  +379.490, Z    +0.000, E1    +0.023, E3 +16426.751}
SPL {X  -159.990, Y  +381.667, Z    +0.000, E1    -4.707, E3 +16426.773}
SPL {X  -159.990, Y  +385.814, Z    +0.000, E1   -15.621, E3 +16426.877}
SPL {X  -159.990, Y  +390.948, Z    +0.000, E1   -28.850, E3 +16427.153}
SPL {X  -159.990, Y  +399.006, Z    +0.000, E1   -45.565, E3 +16427.865}
SPL {X  -159.990, Y  +410.008, Z    +0.000, E1   -58.546, E3 +16429.475}
SPL {X  -159.990, Y  +426.664, Z    +0.000, E1   -66.963, E3 +16433.096}
SPL {X  -159.990, Y  +494.829, Z    +0.000, E1   -73.764, E3 +16454.860}
SPL {X  -158.798, Y  +695.991, Z    +0.000, E1   -74.986, E3 +16544.793}
SPL {X  -156.512, Y  +709.677, Z    +0.000, E1   -74.772, E3 +16554.937}
SPL {X  -153.684, Y  +720.975, Z    +0.000, E1   -74.508, E3 +16564.224}
SPL {X  -150.879, Y  +729.719, Z    +0.000, E1   -74.224, E3 +16572.018}
SPL {X  -148.237, Y  +736.689, Z    +0.000, E1   -73.960, E3 +16578.572}
SPL {X  -145.190, Y  +743.705, Z    +0.000, E1   -73.640, E3 +16585.493}
SPL {X  -141.940, Y  +750.322, Z    +0.000, E1   -73.290, E3 +16592.260}
SPL {X  -138.555, Y  +756.496, Z    +0.000, E1   -72.905, E3 +16598.825}
SPL {X  -135.025, Y  +762.319, Z    +0.000, E1   -72.483, E3 +16605.204}
SPL {X  -131.747, Y  +767.272, Z    +0.000, E1   -72.071, E3 +16610.729}
SPL {X  -127.432, Y  +773.236, Z    +0.000, E1   -71.530, E3 +16617.415}
SPL {X  -124.036, Y  +777.554, Z    +0.000, E1   -71.026, E3 +16622.313}
SPL {X  -120.782, Y  +781.422, Z    +0.000, E1   -70.584, E3 +16626.571}
SPL {X   -74.295, Y  +818.193, Z    +0.000, E1   -57.793, E3 +16736.902}
ENDSPLINE

SPLINE
SPL {X  -105.102, Y  +797.125, Z    +0.000, E1   -55.734, E3 +16916.268}
SPL {X  -126.361, Y  +774.631, Z    +0.000, E1   -54.192, E3 +16941.936}
SPL {X  -145.777, Y  +742.423, Z    +0.000, E1   -46.722, E3 +16957.277}
SPL {X  -154.920, Y  +716.458, Z    +0.000, E1   -35.175, E3 +16963.332}
SPL {X  -158.252, Y  +700.019, Z    +0.000, E1   -24.087, E3 +16965.584}
SPL {X  -159.434, Y  +689.826, Z    +0.000, E1   -15.506, E3 +16966.402}
SPL {X  -159.958, Y  +679.684, Z    +0.000, E1    -5.688, E3 +16966.825}
SPL {X  -159.990, Y  +674.512, Z    +0.000, E1    -0.026, E3 +16966.890}
SPL {X  -159.990, Y  +672.767, Z    +0.000, E1    +3.705, E3 +16966.903}
SPL {X  -159.990, Y  +669.310, Z    +0.000, E1   +12.444, E3 +16966.977}
SPL {X  -159.990, Y  +665.511, Z    +0.000, E1   +22.359, E3 +16967.136}
SPL {X  -159.990, Y  +660.776, Z    +0.000, E1   +34.018, E3 +16967.442}
SPL {X  -159.990, Y  +655.863, Z    +0.000, E1   +43.768, E3 +16967.900}
SPL {X  -159.990, Y  +646.280, Z    +0.000, E1   +56.156, E3 +16969.189}
SPL {X  -159.990, Y  +625.549, Z    +0.000, E1   +67.208, E3 +16973.711}
SPL {X  -159.990, Y  +550.186, Z    +0.000, E1   +73.637, E3 +16999.117}
SPL {X  -159.878, Y  +371.520, Z    +0.000, E1   +74.559, E3 +17081.879}
SPL {X  -159.109, Y  +360.737, Z    +0.000, E1   +74.490, E3 +17089.003}
SPL {X  -156.915, Y  +346.281, Z    +0.000, E1   +74.304, E3 +17099.706}
ENDSPLINE

SPLINE
SPL {X  -159.697, Y  +367.814, Z    +0.000, E1   +71.217, E3 +17117.024}
ENDSPLINE

SPLINE
SPL {X  -156.028, Y  +342.114, Z    +0.000, E1   +72.020, E3 +17127.178}
SPL {X  -150.925, Y  +324.412, Z    +0.000, E1   +72.419, E3 +17134.971}
SPL {X  -144.972, Y  +309.824, Z    +0.000, E1   +72.799, E3 +17140.573}
SPL {X  -139.605, Y  +299.351, Z    +0.000, E1   +73.035, E3 +17144.704}
SPL {X  -136.475, Y  +294.006, Z    +0.000, E1   +72.670, E3 +17150.489}
SPL {X  -133.214, Y  +288.895, Z    +0.000, E1   +72.272, E3 +17156.137}
SPL {X  -129.829, Y  +284.006, Z    +0.000, E1   +71.844, E3 +17161.612}
SPL {X  -125.428, Y  +278.179, Z    +0.000, E1   +71.273, E3 +17168.149}
SPL {X  -120.729, Y  +272.518, Z    +0.000, E1   +70.593, E3 +17174.459}
SPL {X   -77.409, Y  +237.483, Z    +0.000, E1   +59.013, E3 +17269.310}
ENDSPLINE

SPLINE
SPL {X  -103.775, Y  +255.731, Z    +0.000, E1   +56.205, E3 +17466.023}
SPL {X  -141.196, Y  +302.265, Z    +0.000, E1   +49.914, E3 +17503.508}
SPL {X  -153.296, Y  +331.706, Z    +0.000, E1   +38.681, E3 +17511.927}
SPL {X  -157.534, Y  +349.577, Z    +0.000, E1   +27.748, E3 +17514.555}
SPL {X  -159.460, Y  +364.489, Z    +0.000, E1   +15.407, E3 +17515.850}
SPL {X  -159.962, Y  +374.520, Z    +0.000, E1    +5.534, E3 +17516.246}
SPL {X  -159.990, Y  +379.490, Z    +0.000, E1    +0.023, E3 +17516.303}
SPL {X  -159.990, Y  +381.667, Z    +0.000, E1    -4.707, E3 +17516.325}
SPL {X  -159.990, Y  +387.434, Z    +0.000, E1   -19.600, E3 +17516.508}
SPL {X  -159.990, Y  +392.971, Z    +0.000, E1   -33.903, E3 +17516.841}
SPL {X  -159.990, Y  +399.006, Z    +0.000, E1   -45.565, E3 +17517.417}
SPL {X  -159.990, Y  +410.008, Z    +0.000, E1   -58.546, E3 +17519.027}
SPL {X  -159.990, Y  +426.664, Z    +0.000, E1   -66.963, E3 +17522.649}
SPL {X  -159.990, Y  +494.829, Z    +0.000, E1   -73.764, E3 +17544.413}
SPL {X  -158.798, Y  +695.991, Z    +0.000, E1   -74.986, E3 +17634.345}
SPL {X  -156.512, Y  +709.677, Z    +0.000, E1   -74.772, E3 +17644.489}
SPL {X  -153.684, Y  +720.975, Z    +0.000, E1   -74.508, E3 +17653.776}
SPL {X  -149.353, Y  +733.863, Z    +0.000, E1   -74.100, E3 +17665.364}
SPL {X  -145.190, Y  +743.705, Z    +0.000, E1   -73.640, E3 +17675.045}
SPL {X  -141.940, Y  +750.322, Z    +0.000, E1   -73.290, E3 +17681.812}
SPL {X  -138.555, Y  +756.496, Z    +0.000, E1   -72.905, E3 +17688.377}
SPL {X  -135.025, Y  +762.319, Z    +0.000, E1   -72.483, E3 +17694.756}
SPL {X  -131.747, Y  +767.272, Z    +0.000, E1   -72.071, E3 +17700.281}
SPL {X  -127.432, Y  +773.236, Z    +0.000, E1   -71.530, E3 +17706.967}
SPL {X  -124.036, Y  +777.554, Z    +0.000, E1   -71.026, E3 +17711.865}
SPL {X  -120.782, Y  +781.422, Z    +0.000, E1   -70.584, E3 +17716.123}
SPL {X   -74.295, Y  +818.193, Z    +0.000, E1   -57.793, E3 +17826.454}
ENDSPLINE

SPLINE
SPL {X  -120.240, Y  +782.043, Z    +0.000, E1   -55.019, E3 +18024.950}
SPL {X  -145.777, Y  +742.423, Z    +0.000, E1   -46.722, E3 +18046.829}
SPL {X  -154.920, Y  +716.458, Z    +0.000, E1   -35.175, E3 +18052.884}
SPL {X  -158.252, Y  +700.019, Z    +0.000, E1   -24.087, E3 +18055.136}
SPL {X  -159.676, Y  +686.525, Z    +0.000, E1   -12.514, E3 +18056.126}
SPL {X  -159.990, Y  +674.678, Z    +0.000, E1    -0.382, E3 +18056.441}
SPL {X  -159.990, Y  +672.767, Z    +0.000, E1    +3.705, E3 +18056.455}
SPL {X  -159.990, Y  +669.310, Z    +0.000, E1   +12.444, E3 +18056.529}
SPL {X  -159.990, Y  +665.511, Z    +0.000, E1   +22.359, E3 +18056.688}
SPL {X  -159.990, Y  +658.432, Z    +0.000, E1   +38.720, E3 +18057.213}
SPL {X  -159.990, Y  +646.280, Z    +0.000, E1   +56.156, E3 +18058.741}
SPL {X  -159.990, Y  +625.549, Z    +0.000, E1   +67.208, E3 +18063.263}
SPL {X  -159.990, Y  +550.186, Z    +0.000, E1   +73.637, E3 +18088.669}
SPL {X  -159.878, Y  +371.520, Z    +0.000, E1   +74.559, E3 +18171.431}
SPL {X  -158.372, Y  +354.804, Z    +0.000, E1   +74.445, E3 +18182.735}
SPL {X  -156.009, Y  +342.031, Z    +0.000, E1   +74.195, E3 +18192.745}
ENDSPLINE

SPLINE
SPL {X  -159.697, Y  +367.814, Z    +0.000, E1   +71.217, E3 +18206.577}
ENDSPLINE

SPLINE
SPL {X  -156.028, Y  +342.114, Z    +0.000, E1   +72.020, E3 +18216.730}
SPL {X  -150.925, Y  +324.412, Z    +0.000, E1   +72.419, E3 +18224.523}
SPL {X  -144.972, Y  +309.824, Z    +0.000, E1   +72.799, E3 +18230.125}
SPL {X  -139.605, Y  +299.351, Z    +0.000, E1   +73.035, E3 +18234.257}
SPL {X  -136.475, Y  +294.006, Z    +0.000, E1   +72.670, E3 +18240.042}
SPL {X  -133.214, Y  +288.895, Z    +0.000, E1   +72.272, E3 +18245.689}
SPL {X  -129.829, Y  +284.006, Z    +0.000, E1   +71.844, E3 +18251.164}
SPL {X  -125.428, Y  +278.179, Z    +0.000, E1   +71.273, E3 +18257.702}
SPL {X  -120.729, Y  +272.518, Z    +0.000, E1   +70.593, E3 +18264.011}
SPL {X   -77.409, Y  +237.483, Z    +0.000, E1   +59.013, E3 +18358.862}
ENDSPLINE

SPLINE
SPL {X  -103.775, Y  +255.731, Z    +0.000, E1   +56.205, E3 +18555.575}
SPL {X  -133.021, Y  +288.605, Z    +0.000, E1   +53.007, E3 +18587.032}
SPL {X  -149.384, Y  +320.219, Z    +0.000, E1   +43.953, E3 +18598.755}
SPL {X  -157.534, Y  +349.577, Z    +0.000, E1   +27.748, E3 +18604.107}
SPL {X  -159.460, Y  +364.489, Z    +0.000, E1   +15.407, E3 +18605.403}
SPL {X  -159.962, Y  +374.520, Z    +0.000, E1    +5.534, E3 +18605.798}
SPL {X  -159.990, Y  +379.741, Z    +0.000, E1    -0.257, E3 +18605.857}
SPL {X  -159.990, Y  +384.604, Z    +0.000, E1   -12.124, E3 +18605.946}
SPL {X  -159.990, Y  +389.475, Z    +0.000, E1   -25.351, E3 +18606.159}
SPL {X  -159.990, Y  +395.000, Z    +0.000, E1   -38.121, E3 +18606.569}
SPL {X  -159.990, Y  +406.380, Z    +0.000, E1   -55.108, E3 +18608.011}
SPL {X  -159.990, Y  +426.664, Z    +0.000, E1   -66.963, E3 +18612.201}
SPL {X  -159.990, Y  +494.829, Z    +0.000, E1   -73.764, E3 +18633.965}
SPL {X  -158.798, Y  +695.991, Z    +0.000, E1   -74.986, E3 +18723.898}
SPL {X  -156.512, Y  +709.677, Z    +0.000, E1   -74.772, E3 +18734.041}
SPL {X  -153.684, Y  +720.975, Z    +0.000, E1   -74.508, E3 +18743.329}
SPL {X  -149.353, Y  +733.863, Z    +0.000, E1   -74.100, E3 +18754.916}
SPL {X  -145.190, Y  +743.705, Z    +0.000, E1   -73.640, E3 +18764.597}
SPL {X  -141.940, Y  +750.322, Z    +0.000, E1   -73.290, E3 +18771.364}
SPL {X  -138.555, Y  +756.496, Z    +0.000, E1   -72.905, E3 +18777.929}
SPL {X  -135.025, Y  +762.319, Z    +0.000, E1   -72.483, E3 +18784.309}
SPL {X  -131.747, Y  +767.272, Z    +0.000, E1   -72.071, E3 +18789.834}
SPL {X  -127.432, Y  +773.236, Z    +0.000, E1   -71.530, E3 +18796.519}
SPL {X  -124.036, Y  +777.554, Z    +0.000, E1   -71.026, E3 +18801.418}
SPL {X  -120.782, Y  +781.422, Z    +0.000, E1   -70.584, E3 +18805.675}
SPL {X   -74.295, Y  +818.193, Z    +0.000, E1   -57.793, E3 +18916.006}
ENDSPLINE

SPLINE
SPL {X  -120.240, Y  +782.043, Z    +0.000, E1   -55.019, E3 +19114.502}
SPL {X  -145.777, Y  +742.423, Z    +0.000, E1   -46.722, E3 +19136.381}
SPL {X  -154.920, Y  +716.458, Z    +0.000, E1   -35.175, E3 +19142.436}
SPL {X  -158.252, Y  +700.019, Z    +0.000, E1   -24.087, E3 +19144.688}
SPL {X  -159.676, Y  +686.525, Z    +0.000, E1   -12.514, E3 +19145.678}
SPL {X  -159.990, Y  +674.678, Z    +0.000, E1    -0.382, E3 +19145.993}
SPL {X  -159.990, Y  +672.767, Z    +0.000, E1    +3.705, E3 +19146.008}
SPL {X  -159.990, Y  +669.310, Z    +0.000, E1   +12.444, E3 +19146.081}
SPL {X  -159.990, Y  +665.511, Z    +0.000, E1   +22.359, E3 +19146.240}
SPL {X  -159.990, Y  +660.776, Z    +0.000, E1   +34.018, E3 +19146.547}
SPL {X  -159.990, Y  +655.863, Z    +0.000, E1   +43.768, E3 +19147.004}
SPL {X  -159.990, Y  +646.280, Z    +0.000, E1   +56.156, E3 +19148.294}
SPL {X  -159.990, Y  +625.549, Z    +0.000, E1   +67.208, E3 +19152.815}
SPL {X  -159.990, Y  +550.186, Z    +0.000, E1   +73.637, E3 +19178.221}
SPL {X  -159.878, Y  +371.520, Z    +0.000, E1   +74.559, E3 +19260.983}
SPL {X  -159.109, Y  +360.737, Z    +0.000, E1   +74.490, E3 +19268.107}
SPL {X  -156.915, Y  +346.281, Z    +0.000, E1   +74.304, E3 +19278.810}
ENDSPLINE

SPLINE
SPL {X  -159.697, Y  +367.814, Z    +0.000, E1   +71.217, E3 +19296.129}
ENDSPLINE

SPLINE
SPL {X  -156.028, Y  +342.114, Z    +0.000, E1   +72.020, E3 +19306.282}
SPL {X  -150.925, Y  +324.412, Z    +0.000, E1   +72.419, E3 +19314.075}
SPL {X  -146.819, Y  +313.931, Z    +0.000, E1   +72.621, E3 +19318.768}
SPL {X  -140.820, Y  +301.561, Z    +0.000, E1   +73.023, E3 +19322.685}
SPL {X  -136.475, Y  +294.006, Z    +0.000, E1   +72.670, E3 +19329.594}
SPL {X  -133.214, Y  +288.895, Z    +0.000, E1   +72.272, E3 +19335.242}
SPL {X  -129.829, Y  +284.006, Z    +0.000, E1   +71.844, E3 +19340.716}
SPL {X  -125.428, Y  +278.179, Z    +0.000, E1   +71.273, E3 +19347.254}
SPL {X  -120.729, Y  +272.518, Z    +0.000, E1   +70.593, E3 +19353.563}
SPL {X   -77.409, Y  +237.483, Z    +0.000, E1   +59.013, E3 +19448.414}
ENDSPLINE

SPLINE
SPL {X  -103.775, Y  +255.731, Z    +0.000, E1   +56.205, E3 +19645.127}
SPL {X  -141.196, Y  +302.265, Z    +0.000, E1   +49.914, E3 +19682.613}
SPL {X  -155.405, Y  +339.473, Z    +0.000, E1   +34.418, E3 +19692.313}
SPL {X  -159.172, Y  +361.346, Z    +0.000, E1   +18.323, E3 +19694.738}
SPL {X  -159.962, Y  +374.520, Z    +0.000, E1    +5.534, E3 +19695.350}
SPL {X  -159.990, Y  +379.490, Z    +0.000, E1    +0.023, E3 +19695.408}
SPL {X  -159.990, Y  +381.667, Z    +0.000, E1    -4.707, E3 +19695.430}
SPL {X  -159.990, Y  +385.814, Z    +0.000, E1   -15.621, E3 +19695.534}
SPL {X  -159.990, Y  +390.948, Z    +0.000, E1   -28.850, E3 +19695.810}
SPL {X  -159.990, Y  +399.006, Z    +0.000, E1   -45.565, E3 +19696.522}
SPL {X  -159.990, Y  +410.008, Z    +0.000, E1   -58.546, E3 +19698.132}
SPL {X  -159.990, Y  +426.664, Z    +0.000, E1   -66.963, E3 +19701.753}
SPL {X  -159.990, Y  +494.829, Z    +0.000, E1   -73.764, E3 +19723.517}
SPL {X  -158.798, Y  +695.991, Z    +0.000, E1   -74.986, E3 +19813.450}
SPL {X  -156.512, Y  +709.677, Z    +0.000, E1   -74.772, E3 +19823.593}
SPL {X  -153.684, Y  +720.975, Z    +0.000, E1   -74.508, E3 +19832.881}
SPL {X  -149.353, Y  +733.863, Z    +0.000, E1   -74.100, E3 +19844.468}
SPL {X  -145.190, Y  +743.705, Z    +0.000, E1   -73.640, E3 +19854.150}
SPL {X  -141.940, Y  +750.322, Z    +0.000, E1   -73.290, E3 +19860.916}
SPL {X  -138.555, Y  +756.496, Z    +0.000, E1   -72.905, E3 +19867.481}
SPL {X  -135.025, Y  +762.319, Z    +0.000, E1   -72.483, E3 +19873.861}
SPL {X  -131.747, Y  +767.272, Z    +0.000, E1   -72.071, E3 +19879.386}
SPL {X  -127.432, Y  +773.236, Z    +0.000, E1   -71.530, E3 +19886.071}
SPL {X  -124.036, Y  +777.554, Z    +0.000, E1   -71.026, E3 +19890.970}
SPL {X  -120.782, Y  +781.422, Z    +0.000, E1   -70.584, E3 +19895.228}
SPL {X   -74.295, Y  +818.193, Z    +0.000, E1   -57.793, E3 +20005.558}
ENDSPLINE

SPLINE
SPL {X  -105.102, Y  +797.125, Z    +0.000, E1   -55.734, E3 +20184.925}
SPL {X  -126.361, Y  +774.631, Z    +0.000, E1   -54.192, E3 +20210.593}
SPL {X  -145.777, Y  +742.423, Z    +0.000, E1   -46.722, E3 +20225.934}
SPL {X  -154.920, Y  +716.458, Z    +0.000, E1   -35.175, E3 +20231.989}
SPL {X  -159.063, Y  +693.702, Z    +0.000, E1   -19.028, E3 +20234.770}
SPL {X  -159.958, Y  +679.684, Z    +0.000, E1    -5.688, E3 +20235.482}
SPL {X  -159.990, Y  +674.512, Z    +0.000, E1    -0.026, E3 +20235.546}
SPL {X  -159.990, Y  +672.767, Z    +0.000, E1    +3.705, E3 +20235.560}
SPL {X  -159.990, Y  +669.310, Z    +0.000, E1   +12.444, E3 +20235.634}
SPL {X  -159.990, Y  +665.511, Z    +0.000, E1   +22.359, E3 +20235.792}
SPL {X  -159.990, Y  +658.432, Z    +0.000, E1   +38.720, E3 +20236.317}
SPL {X  -159.990, Y  +646.280, Z    +0.000, E1   +56.156, E3 +20237.846}
SPL {X  -159.990, Y  +625.549, Z    +0.000, E1   +67.208, E3 +20242.368}
SPL {X  -159.990, Y  +550.186, Z    +0.000, E1   +73.637, E3 +20267.773}
SPL {X  -159.878, Y  +371.520, Z    +0.000, E1   +74.559, E3 +20350.535}
SPL {X  -159.109, Y  +360.737, Z    +0.000, E1   +74.490, E3 +20357.660}
SPL {X  -156.915, Y  +346.281, Z    +0.000, E1   +74.304, E3 +20368.363}
ENDSPLINE

SPLINE
SPL {X  -159.697, Y  +367.814, Z    +0.000, E1   +71.217, E3 +20385.681}
ENDSPLINE

SPLINE
SPL {X  -156.028, Y  +342.114, Z    +0.000, E1   +72.020, E3 +20395.835}
SPL {X  -150.925, Y  +324.412, Z    +0.000, E1   +72.419, E3 +20403.627}
SPL {X  -144.972, Y  +309.824, Z    +0.000, E1   +72.799, E3 +20409.229}
SPL {X  -139.605, Y  +299.351, Z    +0.000, E1   +73.035, E3 +20413.361}
SPL {X  -136.475, Y  +294.006, Z    +0.000, E1   +72.670, E3 +20419.146}
SPL {X  -133.214, Y  +288.895, Z    +0.000, E1   +72.272, E3 +20424.794}
SPL {X  -129.829, Y  +284.006, Z    +0.000, E1   +71.844, E3 +20430.269}
SPL {X  -125.428, Y  +278.179, Z    +0.000, E1   +71.273, E3 +20436.806}
SPL {X  -120.729, Y  +272.518, Z    +0.000, E1   +70.593, E3 +20443.115}
SPL {X   -77.409, Y  +237.483, Z    +0.000, E1   +59.013, E3 +20537.966}
ENDSPLINE

SPLINE
SPL {X  -103.775, Y  +255.731, Z    +0.000, E1   +56.205, E3 +20734.680}
SPL {X  -141.196, Y  +302.265, Z    +0.000, E1   +49.914, E3 +20772.165}
SPL {X  -155.405, Y  +339.473, Z    +0.000, E1   +34.418, E3 +20781.865}
SPL {X  -159.172, Y  +361.346, Z    +0.000, E1   +18.323, E3 +20784.290}
SPL {X  -159.962, Y  +374.520, Z    +0.000, E1    +5.534, E3 +20784.903}
SPL {X  -159.990, Y  +379.490, Z    +0.000, E1    +0.023, E3 +20784.960}
SPL {X  -159.990, Y  +381.667, Z    +0.000, E1    -4.707, E3 +20784.982}
SPL {X  -159.990, Y  +385.814, Z    +0.000, E1   -15.621, E3 +20785.086}
SPL {X  -159.990, Y  +390.948, Z    +0.000, E1   -28.850, E3 +20785.362}
SPL {X  -159.990, Y  +399.006, Z    +0.000, E1   -45.565, E3 +20786.074}
SPL {X  -159.990, Y  +410.008, Z    +0.000, E1   -58.546, E3 +20787.684}
SPL {X  -159.990, Y  +426.664, Z    +0.000, E1   -66.963, E3 +20791.305}
SPL {X  -159.990, Y  +494.829, Z    +0.000, E1   -73.764, E3 +20813.069}
SPL {X  -158.798, Y  +695.991, Z    +0.000, E1   -74.986, E3 +20903.002}
SPL {X  -156.512, Y  +709.677, Z    +0.000, E1   -74.772, E3 +20913.146}
SPL {X  -153.684, Y  +720.975, Z    +0.000, E1   -74.508, E3 +20922.433}
SPL {X  -149.353, Y  +733.863, Z    +0.000, E1   -74.100, E3 +20934.021}
SPL {X  -145.190, Y  +743.705, Z    +0.000, E1   -73.640, E3 +20943.702}
SPL {X  -141.940, Y  +750.322, Z    +0.000, E1   -73.290, E3 +20950.469}
SPL {X  -138.555, Y  +756.496, Z    +0.000, E1   -72.905, E3 +20957.034}
SPL {X  -135.025, Y  +762.319, Z    +0.000, E1   -72.483, E3 +20963.413}
SPL {X  -131.747, Y  +767.272, Z    +0.000, E1   -72.071, E3 +20968.938}
SPL {X  -127.432, Y  +773.236, Z    +0.000, E1   -71.530, E3 +20975.624}
SPL {X  -122.390, Y  +779.541, Z    +0.000, E1   -70.825, E3 +20982.698}
SPL {X  -119.460, Y  +782.925, Z    +0.000, E1   -70.353, E3 +20986.450}
SPL {X   -74.295, Y  +818.193, Z    +0.000, E1   -57.793, E3 +21095.111}
ENDSPLINE

SPLINE
SPL {X  -120.240, Y  +782.043, Z    +0.000, E1   -55.019, E3 +21293.606}
SPL {X  -145.777, Y  +742.423, Z    +0.000, E1   -46.722, E3 +21315.486}
SPL {X  -154.920, Y  +716.458, Z    +0.000, E1   -35.175, E3 +21321.541}
SPL {X  -158.252, Y  +700.019, Z    +0.000, E1   -24.087, E3 +21323.793}
SPL {X  -159.434, Y  +689.826, Z    +0.000, E1   -15.506, E3 +21324.611}
SPL {X  -159.958, Y  +679.684, Z    +0.000, E1    -5.688, E3 +21325.034}
SPL {X  -159.990, Y  +674.512, Z    +0.000, E1    -0.026, E3 +21325.099}
SPL {X  -159.990, Y  +672.767, Z    +0.000, E1    +3.705, E3 +21325.112}
SPL {X  -159.990, Y  +669.310, Z    +0.000, E1   +12.444, E3 +21325.186}
SPL {X  -159.990, Y  +665.511, Z    +0.000, E1   +22.359, E3 +21325.345}
SPL {X  -159.990, Y  +658.432, Z    +0.000, E1   +38.720, E3 +21325.870}
SPL {X  -159.990, Y  +646.280, Z    +0.000, E1   +56.156, E3 +21327.398}
SPL {X  -159.990, Y  +625.549, Z    +0.000, E1   +67.208, E3 +21331.920}
SPL {X  -159.990, Y  +550.186, Z    +0.000, E1   +73.637, E3 +21357.326}
SPL {X  -159.493, Y  +364.902, Z    +0.000, E1   +74.541, E3 +21444.319}
SPL {X  -156.915, Y  +346.281, Z    +0.000, E1   +74.304, E3 +21457.915}
ENDSPLINE

SPLINE
SPL {X  -159.697, Y  +367.814, Z    +0.000, E1   +71.217, E3 +21475.233}
ENDSPLINE

SPLINE
SPL {X  -156.028, Y  +342.114, Z    +0.000, E1   +72.020, E3 +21485.387}
SPL {X  -150.925, Y  +324.412, Z    +0.000, E1   +72.419, E3 +21493.180}
SPL {X  -144.972, Y  +309.824, Z    +0.000, E1   +72.799, E3 +21498.782}
SPL {X  -139.605, Y  +299.351, Z    +0.000, E1   +73.035, E3 +21502.913}
SPL {X  -136.475, Y  +294.006, Z    +0.000, E1   +72.670, E3 +21508.698}
SPL {X  -133.214, Y  +288.895, Z    +0.000, E1   +72.272, E3 +21514.346}
SPL {X  -129.829, Y  +284.006, Z    +0.000, E1   +71.844, E3 +21519.821}
SPL {X  -125.428, Y  +278.179, Z    +0.000, E1   +71.273, E3 +21526.358}
SPL {X  -120.729, Y  +272.518, Z    +0.000, E1   +70.593, E3 +21532.668}
SPL {X   -77.409, Y  +237.483, Z    +0.000, E1   +59.013, E3 +21627.519}
ENDSPLINE

SPLINE
SPL {X  -103.775, Y  +255.731, Z    +0.000, E1   +56.205, E3 +21824.232}
SPL {X  -141.196, Y  +302.265, Z    +0.000, E1   +49.914, E3 +21861.717}
SPL {X  -153.296, Y  +331.706, Z    +0.000, E1   +38.681, E3 +21870.136}
SPL {X  -157.534, Y  +349.577, Z    +0.000, E1   +27.748, E3 +21872.764}
SPL {X  -159.460, Y  +364.489, Z    +0.000, E1   +15.407, E3 +21874.059}
SPL {X  -159.962, Y  +374.520, Z    +0.000, E1    +5.534, E3 +21874.455}
SPL {X  -159.990, Y  +379.490, Z    +0.000, E1    +0.023, E3 +21874.512}
SPL {X  -159.990, Y  +381.667, Z    +0.000, E1    -4.707, E3 +21874.534}
SPL {X  -159.990, Y  +385.814, Z    +0.000, E1   -15.621, E3 +21874.638}
SPL {X  -159.990, Y  +390.948, Z    +0.000, E1   -28.850, E3 +21874.914}
SPL {X  -159.990, Y  +399.006, Z    +0.000, E1   -45.565, E3 +21875.626}
SPL {X  -159.990, Y  +410.008, Z    +0.000, E1   -58.546, E3 +21877.236}
SPL {X  -159.990, Y  +430.714, Z    +0.000, E1   -67.965, E3 +21882.042}
SPL {X  -159.990, Y  +500.758, Z    +0.000, E1   -73.927, E3 +21904.717}
SPL {X  -158.798, Y  +695.991, Z    +0.000, E1   -74.986, E3 +21992.554}
SPL {X  -156.512, Y  +709.677, Z    +0.000, E1   -74.772, E3 +22002.698}
SPL {X  -153.684, Y  +720.975, Z    +0.000, E1   -74.508, E3 +22011.985}
SPL {X  -149.353, Y  +733.863, Z    +0.000, E1   -74.100, E3 +22023.573}
SPL {X  -145.190, Y  +743.705, Z    +0.000, E1   -73.640, E3 +22033.254}
SPL {X  -141.940, Y  +750.322, Z    +0.000, E1   -73.290, E3 +22040.021}
SPL {X  -138.555, Y  +756.496, Z    +0.000, E1   -72.905, E3 +22046.586}
SPL {X  -135.025, Y  +762.319, Z    +0.000, E1   -72.483, E3 +22052.965}
SPL {X  -131.747, Y  +767.272, Z    +0.000, E1   -72.071, E3 +22058.490}
SPL {X  -128.648, Y  +771.613, Z    +0.000, E1   -71.666, E3 +22063.383}
SPL {X  -125.012, Y  +776.344, Z    +0.000, E1   -71.184, E3 +22068.694}
SPL {X  -121.578, Y  +780.498, Z    +0.000, E1   -70.681, E3 +22073.338}
SPL {X  -119.460, Y  +782.925, Z    +0.000, E1   -70.353, E3 +22076.002}
SPL {X   -74.295, Y  +818.193, Z    +0.000, E1   -57.793, E3 +22184.663}
ENDSPLINE

SPLINE
SPL {X  -120.240, Y  +782.043, Z    +0.000, E1   -55.019, E3 +22383.159}
SPL {X  -145.777, Y  +742.423, Z    +0.000, E1   -46.722, E3 +22405.038}
SPL {X  -154.920, Y  +716.458, Z    +0.000, E1   -35.175, E3 +22411.093}
SPL {X  -159.063, Y  +693.702, Z    +0.000, E1   -19.028, E3 +22413.874}
SPL {X  -159.958, Y  +679.684, Z    +0.000, E1    -5.688, E3 +22414.586}
SPL {X  -159.990, Y  +674.512, Z    +0.000, E1    -0.026, E3 +22414.651}
SPL {X  -159.990, Y  +672.767, Z    +0.000, E1    +3.705, E3 +22414.664}
SPL {X  -159.990, Y  +669.310, Z    +0.000, E1   +12.444, E3 +22414.738}
SPL {X  -159.990, Y  +665.511, Z    +0.000, E1   +22.359, E3 +22414.897}
SPL {X  -159.990, Y  +658.432, Z    +0.000, E1   +38.720, E3 +22415.422}
SPL {X  -159.990, Y  +646.280, Z    +0.000, E1   +56.156, E3 +22416.950}
SPL {X  -159.990, Y  +625.549, Z    +0.000, E1   +67.208, E3 +22421.472}
SPL {X  -159.990, Y  +550.186, Z    +0.000, E1   +73.637, E3 +22446.878}
SPL {X  -159.493, Y  +364.902, Z    +0.000, E1   +74.541, E3 +22533.871}
SPL {X  -156.915, Y  +346.281, Z    +0.000, E1   +74.304, E3 +22547.467}
ENDSPLINE

SPLINE
SPL {X  -159.697, Y  +367.814, Z    +0.000, E1   +71.217, E3 +22564.786}
ENDSPLINE

SPLINE
SPL {X  -156.028, Y  +342.114, Z    +0.000, E1   +72.020, E3 +22574.939}
SPL {X  -150.925, Y  +324.412, Z    +0.000, E1   +72.419, E3 +22582.732}
SPL {X  -144.972, Y  +309.824, Z    +0.000, E1   +72.799, E3 +22588.334}
SPL {X  -139.605, Y  +299.351, Z    +0.000, E1   +73.035, E3 +22592.466}
SPL {X  -136.475, Y  +294.006, Z    +0.000, E1   +72.670, E3 +22598.250}
SPL {X  -133.214, Y  +288.895, Z    +0.000, E1   +72.272, E3 +22603.898}
SPL {X  -129.829, Y  +284.006, Z    +0.000, E1   +71.844, E3 +22609.373}
SPL {X  -126.314, Y  +279.309, Z    +0.000, E1   +71.374, E3 +22614.665}
SPL {X  -122.705, Y  +274.834, Z    +0.000, E1   +70.869, E3 +22619.677}
SPL {X  -119.804, Y  +271.463, Z    +0.000, E1   +70.429, E3 +22623.395}
SPL {X   -77.409, Y  +237.483, Z    +0.000, E1   +59.013, E3 +22717.071}
ENDSPLINE

SPLINE
SPL {X  -103.775, Y  +255.731, Z    +0.000, E1   +56.205, E3 +22913.784}
SPL {X  -133.021, Y  +288.605, Z    +0.000, E1   +53.007, E3 +22945.241}
SPL {X  -149.384, Y  +320.219, Z    +0.000, E1   +43.953, E3 +22956.964}
SPL {X  -157.534, Y  +349.577, Z    +0.000, E1   +27.748, E3 +22962.316}
SPL {X  -159.460, Y  +364.489, Z    +0.000, E1   +15.407, E3 +22963.611}
SPL {X  -159.962, Y  +374.520, Z    +0.000, E1    +5.534, E3 +22964.007}
SPL {X  -159.990, Y  +379.490, Z    +0.000, E1    +0.023, E3 +22964.065}
SPL {X  -159.990, Y  +381.667, Z    +0.000, E1    -4.707, E3 +22964.087}
SPL {X  -159.990, Y  +387.434, Z    +0.000, E1   -19.600, E3 +22964.269}
SPL {X  -159.990, Y  +392.971, Z    +0.000, E1   -33.903, E3 +22964.602}
SPL {X  -159.990, Y  +399.006, Z    +0.000, E1   -45.565, E3 +22965.178}
SPL {X  -159.990, Y  +410.008, Z    +0.000, E1   -58.546, E3 +22966.789}
SPL {X  -159.990, Y  +426.664, Z    +0.000, E1   -66.963, E3 +22970.410}
SPL {X  -159.990, Y  +494.829, Z    +0.000, E1   -73.764, E3 +22992.174}
SPL {X  -158.798, Y  +695.991, Z    +0.000, E1   -74.986, E3 +23082.107}
SPL {X  -156.512, Y  +709.677, Z    +0.000, E1   -74.772, E3 +23092.250}
SPL {X  -153.684, Y  +720.975, Z    +0.000, E1   -74.508, E3 +23101.537}
SPL {X  -149.353, Y  +733.863, Z    +0.000, E1   -74.100, E3 +23113.125}
SPL {X  -145.190, Y  +743.705, Z    +0.000, E1   -73.640, E3 +23122.806}
SPL {X  -141.940, Y  +750.322, Z    +0.000, E1   -73.290, E3 +23129.573}
SPL {X  -138.555, Y  +756.496, Z    +0.000, E1   -72.905, E3 +23136.138}
SPL {X  -135.025, Y  +762.319, Z    +0.000, E1   -72.483, E3 +23142.518}
SPL {X  -131.747, Y  +767.272, Z    +0.000, E1   -72.071, E3 +23148.043}
SPL {X  -128.648, Y  +771.613, Z    +0.000, E1   -71.666, E3 +23152.935}
SPL {X  -125.012, Y  +776.344, Z    +0.000, E1   -71.184, E3 +23158.247}
SPL {X  -120.782, Y  +781.422, Z    +0.000, E1   -70.584, E3 +23163.884}
SPL {X   -74.295, Y  +818.193, Z    +0.000, E1   -57.793, E3 +23274.215}
ENDSPLINE

SPLINE
SPL {X  -105.102, Y  +797.125, Z    +0.000, E1   -55.734, E3 +23453.582}
SPL {X  -126.361, Y  +774.631, Z    +0.000, E1   -54.192, E3 +23479.249}
SPL {X  -145.777, Y  +742.423, Z    +0.000, E1   -46.722, E3 +23494.590}
SPL {X  -154.920, Y  +716.458, Z    +0.000, E1   -35.175, E3 +23500.645}
SPL {X  -158.252, Y  +700.019, Z    +0.000, E1   -24.087, E3 +23502.897}
SPL {X  -159.676, Y  +686.525, Z    +0.000, E1   -12.514, E3 +23503.887}
SPL {X  -159.990, Y  +674.678, Z    +0.000, E1    -0.382, E3 +23504.202}
SPL {X  -159.990, Y  +672.767, Z    +0.000, E1    +3.705, E3 +23504.216}
SPL {X  -159.990, Y  +669.310, Z    +0.000, E1   +12.444, E3 +23504.290}
SPL {X  -159.990, Y  +665.511, Z    +0.000, E1   +22.359, E3 +23504.449}
SPL {X  -159.990, Y  +658.432, Z    +0.000, E1   +38.720, E3 +23504.974}
SPL {X  -159.990, Y  +646.280, Z    +0.000, E1   +56.156, E3 +23506.503}
SPL {X  -159.990, Y  +625.549, Z    +0.000, E1   +67.208, E3 +23511.024}
SPL {X  -159.990, Y  +550.186, Z    +0.000, E1   +73.637, E3 +23536.430}
SPL {X  -159.878, Y  +371.520, Z    +0.000, E1   +74.559, E3 +23619.192}
SPL {X  -159.109, Y  +360.737, Z    +0.000, E1   +74.490, E3 +23626.316}
SPL {X  -156.915, Y  +346.281, Z    +0.000, E1   +74.304, E3 +23637.019}
ENDSPLINE

SPLINE
SPL {X  -159.697, Y  +367.814, Z    +0.000, E1   +71.217, E3 +23654.338}
ENDSPLINE

SPLINE
SPL {X  -156.028, Y  +342.114, Z    +0.000, E1   +72.020, E3 +23664.491}
SPL {X  -150.925, Y  +324.412, Z    +0.000, E1   +72.419, E3 +23672.284}
SPL {X  -144.972, Y  +309.824, Z    +0.000, E1   +72.799, E3 +23677.886}
SPL {X  -139.605, Y  +299.351, Z    +0.000, E1   +73.035, E3 +23682.018}
SPL {X  -136.475, Y  +294.006, Z    +0.000, E1   +72.670, E3 +23687.803}
SPL {X  -133.214, Y  +288.895, Z    +0.000, E1   +72.272, E3 +23693.450}
SPL {X  -129.829, Y  +284.006, Z    +0.000, E1   +71.844, E3 +23698.925}
SPL {X  -126.314, Y  +279.309, Z    +0.000, E1   +71.374, E3 +23704.218}
SPL {X  -122.705, Y  +274.834, Z    +0.000, E1   +70.869, E3 +23709.229}
SPL {X  -119.804, Y  +271.463, Z    +0.000, E1   +70.429, E3 +23712.948}
SPL {X   -77.409, Y  +237.483, Z    +0.000, E1   +59.013, E3 +23806.623}
ENDSPLINE

SPLINE
SPL {X  -103.775, Y  +255.731, Z    +0.000, E1   +56.205, E3 +24003.336}
SPL {X  -141.196, Y  +302.265, Z    +0.000, E1   +49.914, E3 +24040.821}
SPL {X  -153.296, Y  +331.706, Z    +0.000, E1   +38.681, E3 +24049.241}
SPL {X  -157.534, Y  +349.577, Z    +0.000, E1   +27.748, E3 +24051.868}
SPL {X  -159.460, Y  +364.489, Z    +0.000, E1   +15.407, E3 +24053.164}
SPL {X  -159.962, Y  +374.520, Z    +0.000, E1    +5.534, E3 +24053.559}
SPL {X  -159.990, Y  +379.490, Z    +0.000, E1    +0.023, E3 +24053.617}
SPL {X  -159.990, Y  +381.667, Z    +0.000, E1    -4.707, E3 +24053.639}
SPL {X  -159.990, Y  +387.434, Z    +0.000, E1   -19.600, E3 +24053.821}
SPL {X  -159.990, Y  +392.971, Z    +0.000, E1   -33.903, E3 +24054.154}
SPL {X  -159.990, Y  +399.006, Z    +0.000, E1   -45.565, E3 +24054.731}
SPL {X  -159.990, Y  +410.008, Z    +0.000, E1   -58.546, E3 +24056.341}
SPL {X  -159.990, Y  +426.664, Z    +0.000, E1   -66.963, E3 +24059.962}
SPL {X  -159.990, Y  +494.829, Z    +0.000, E1   -73.764, E3 +24081.726}
SPL {X  -158.798, Y  +695.991, Z    +0.000, E1   -74.986, E3 +24171.659}
SPL {X  -156.512, Y  +709.677, Z    +0.000, E1   -74.772, E3 +24181.802}
SPL {X  -153.684, Y  +720.975, Z    +0.000, E1   -74.508, E3 +24191.090}
SPL {X  -149.353, Y  +733.863, Z    +0.000, E1   -74.100, E3 +24202.677}
SPL {X  -145.190, Y  +743.705, Z    +0.000, E1   -73.640, E3 +24212.359}
SPL {X  -141.940, Y  +750.322, Z    +0.000, E1   -73.290, E3 +24219.125}
SPL {X  -138.555, Y  +756.496, Z    +0.000, E1   -72.905, E3 +24225.690}
SPL {X  -135.025, Y  +762.319, Z    +0.000, E1   -72.483, E3 +24232.070}
SPL {X  -131.747, Y  +767.272, Z    +0.000, E1   -72.071, E3 +24237.595}
SPL {X  -128.648, Y  +771.613, Z    +0.000, E1   -71.666, E3 +24242.487}
SPL {X  -125.012, Y  +776.344, Z    +0.000, E1   -71.184, E3 +24247.799}
SPL {X  -120.782, Y  +781.422, Z    +0.000, E1   -70.584, E3 +24253.437}
SPL {X   -74.295, Y  +818.193, Z    +0.000, E1   -57.793, E3 +24363.767}
ENDSPLINE

SPLINE
SPL {X  -120.240, Y  +782.043, Z    +0.000, E1   -55.019, E3 +24562.263}
SPL {X  -145.777, Y  +742.423, Z    +0.000, E1   -46.722, E3 +24584.142}
SPL {X  -154.920, Y  +716.458, Z    +0.000, E1   -35.175, E3 +24590.197}
SPL {X  -158.252, Y  +700.019, Z    +0.000, E1   -24.087, E3 +24592.449}
SPL {X  -159.434, Y  +689.826, Z    +0.000, E1   -15.506, E3 +24593.268}
SPL {X  -159.958, Y  +679.684, Z    +0.000, E1    -5.688, E3 +24593.691}
SPL {X  -159.990, Y  +674.512, Z    +0.000, E1    -0.026, E3 +24593.755}
SPL {X  -159.990, Y  +672.767, Z    +0.000, E1    +3.705, E3 +24593.769}
SPL {X  -159.990, Y  +669.310, Z    +0.000, E1   +12.444, E3 +24593.843}
SPL {X  -159.990, Y  +665.511, Z    +0.000, E1   +22.359, E3 +24594.001}
SPL {X  -159.990, Y  +658.432, Z    +0.000, E1   +38.720, E3 +24594.526}
SPL {X  -159.990, Y  +646.280, Z    +0.000, E1   +56.156, E3 +24596.055}
SPL {X  -159.990, Y  +625.549, Z    +0.000, E1   +67.208, E3 +24600.576}
SPL {X  -159.990, Y  +550.186, Z    +0.000, E1   +73.637, E3 +24625.982}
SPL {X  -159.493, Y  +364.902, Z    +0.000, E1   +74.541, E3 +24712.975}
SPL {X  -157.674, Y  +350.378, Z    +0.000, E1   +74.357, E3 +24723.432}
SPL {X  -156.009, Y  +342.031, Z    +0.000, E1   +74.195, E3 +24730.059}
ENDSPLINE

SPLINE
SPL {X  -159.697, Y  +367.814, Z    +0.000, E1   +71.217, E3 +24743.890}
ENDSPLINE

SPLINE
SPL {X  -156.028, Y  +342.114, Z    +0.000, E1   +72.020, E3 +24754.044}
SPL {X  -150.925, Y  +324.412, Z    +0.000, E1   +72.419, E3 +24761.836}
SPL {X  -146.819, Y  +313.931, Z    +0.000, E1   +72.621, E3 +24766.530}
SPL {X  -140.820, Y  +301.561, Z    +0.000, E1   +73.023, E3 +24770.446}
SPL {X  -136.475, Y  +294.006, Z    +0.000, E1   +72.670, E3 +24777.355}
SPL {X  -133.214, Y  +288.895, Z    +0.000, E1   +72.272, E3 +24783.003}
SPL {X  -129.829, Y  +284.006, Z    +0.000, E1   +71.844, E3 +24788.478}
SPL {X  -126.314, Y  +279.309, Z    +0.000, E1   +71.374, E3 +24793.770}
SPL {X  -122.705, Y  +274.834, Z    +0.000, E1   +70.869, E3 +24798.781}
SPL {X  -119.804, Y  +271.463, Z    +0.000, E1   +70.429, E3 +24802.500}
SPL {X   -77.409, Y  +237.483, Z    +0.000, E1   +59.013, E3 +24896.175}
ENDSPLINE

SPLINE
SPL {X  -103.775, Y  +255.731, Z    +0.000, E1   +56.205, E3 +25092.889}
SPL {X  -133.021, Y  +288.605, Z    +0.000, E1   +53.007, E3 +25124.345}
SPL {X  -149.384, Y  +320.219, Z    +0.000, E1   +43.953, E3 +25136.068}
SPL {X  -157.534, Y  +349.577, Z    +0.000, E1   +27.748, E3 +25141.420}
SPL {X  -159.460, Y  +364.489, Z    +0.000, E1   +15.407, E3 +25142.716}
SPL {X  -159.962, Y  +374.520, Z    +0.000, E1    +5.534, E3 +25143.112}
SPL {X  -159.990, Y  +379.741, Z    +0.000, E1    -0.257, E3 +25143.170}
SPL {X  -159.990, Y  +384.604, Z    +0.000, E1   -12.124, E3 +25143.259}
SPL {X  -159.990, Y  +390.948, Z    +0.000, E1   -28.850, E3 +25143.571}
SPL {X  -159.990, Y  +399.006, Z    +0.000, E1   -45.565, E3 +25144.283}
SPL {X  -159.990, Y  +410.008, Z    +0.000, E1   -58.546, E3 +25145.893}
SPL {X  -159.990, Y  +426.664, Z    +0.000, E1   -66.963, E3 +25149.514}
SPL {X  -159.990, Y  +494.829, Z    +0.000, E1   -73.764, E3 +25171.278}
SPL {X  -158.798, Y  +695.991, Z    +0.000, E1   -74.986, E3 +25261.211}
SPL {X  -156.512, Y  +709.677, Z    +0.000, E1   -74.772, E3 +25271.355}
SPL {X  -153.684, Y  +720.975, Z    +0.000, E1   -74.508, E3 +25280.642}
SPL {X  -149.353, Y  +733.863, Z    +0.000, E1   -74.100, E3 +25292.230}
SPL {X  -145.190, Y  +743.705, Z    +0.000, E1   -73.640, E3 +25301.911}
SPL {X  -141.940, Y  +750.322, Z    +0.000, E1   -73.290, E3 +25308.678}
SPL {X  -138.555, Y  +756.496, Z    +0.000, E1   -72.905, E3 +25315.243}
SPL {X  -135.025, Y  +762.319, Z    +0.000, E1   -72.483, E3 +25321.622}
SPL {X  -131.747, Y  +767.272, Z    +0.000, E1   -72.071, E3 +25327.147}
SPL {X  -128.648, Y  +771.613, Z    +0.000, E1   -71.666, E3 +25332.039}
SPL {X  -125.012, Y  +776.344, Z    +0.000, E1   -71.184, E3 +25337.351}
SPL {X  -120.782, Y  +781.422, Z    +0.000, E1   -70.584, E3 +25342.989}
SPL {X   -74.295, Y  +818.193, Z    +0.000, E1   -57.793, E3 +25453.320}
ENDSPLINE

SPLINE
SPL {X  -105.102, Y  +797.125, Z    +0.000, E1   -55.734, E3 +25632.686}
SPL {X  -126.361, Y  +774.631, Z    +0.000, E1   -54.192, E3 +25658.354}
SPL {X  -145.777, Y  +742.423, Z    +0.000, E1   -46.722, E3 +25673.695}
SPL {X  -154.920, Y  +716.458, Z    +0.000, E1   -35.175, E3 +25679.750}
SPL {X  -159.063, Y  +693.702, Z    +0.000, E1   -19.028, E3 +25682.531}
SPL {X  -159.958, Y  +679.684, Z    +0.000, E1    -5.688, E3 +25683.243}
SPL {X  -159.990, Y  +674.512, Z    +0.000, E1    -0.026, E3 +25683.308}
SPL {X  -159.990, Y  +672.767, Z    +0.000, E1    +3.705, E3 +25683.321}
SPL {X  -159.990, Y  +669.310, Z    +0.000, E1   +12.444, E3 +25683.395}
SPL {X  -159.990, Y  +665.511, Z    +0.000, E1   +22.359, E3 +25683.554}
SPL {X  -159.990, Y  +660.776, Z    +0.000, E1   +34.018, E3 +25683.860}
SPL {X  -159.990, Y  +655.863, Z    +0.000, E1   +43.768, E3 +25684.318}
SPL {X  -159.990, Y  +646.280, Z    +0.000, E1   +56.156, E3 +25685.607}
SPL {X  -159.990, Y  +625.549, Z    +0.000, E1   +67.208, E3 +25690.129}
SPL {X  -159.990, Y  +550.186, Z    +0.000, E1   +73.637, E3 +25715.534}
SPL {X  -159.493, Y  +364.902, Z    +0.000, E1   +74.541, E3 +25802.528}
SPL {X  -156.915, Y  +346.281, Z    +0.000, E1   +74.304, E3 +25816.124}
ENDSPLINE

SPLINE
SPL {X  -159.697, Y  +367.814, Z    +0.000, E1   +71.217, E3 +25833.442}
ENDSPLINE

